(* CoDeSys 2.3.9.59 project: 4.2_Engine_Safety_System20170112.pro *)
(* Libraries: WagoLibTerminalDiag.lib 8.11.10 10:37:48, SYSLIBMEM.LIB 8.11.10 10:37:48, SysLibRtc.lib 8.11.10 10:37:48, Util.lib 26.9.14 11:12:46, WagoLib_CAN_Gateway_02.lib*21.5.19 15:49:18, WagoLibMBX_01.lib*23.7.19 16:23:10, WagoLibMBX_System_01.lib*10.7.18 13:47:36, Standard.lib 8.11.10 10:37:48, SYSLIBCALLBACK.LIB 8.11.10 10:37:48, WagoLibSockets.lib 14.5.12 10:49:54, SysLibSockets.lib 5.5.11 07:22:24, NETVARUDP_LIB_V23.LIB*29.6.15 15:12:14, WagoLibModbus_IP_01.lib*11.2.19 15:41:00, Wago_MBCFG_ETHERNET_01.lib*10.7.18 13:47:36, Wago_MBCFG_COMMON_01.lib*10.7.18 13:47:36 *)

(* PLC configuration (modules and I/O channels)
0750-1504 16 DO 24V DC 0.5A [Type_10_16_Channels] node 0, in %IB36 out %QB36 {INTTypePAAssignment = PLC; INTTypeModule = plugged}
  AT %QX18.0 [BOOLOnX_Q] Ch_1 Digital output
  AT %QX18.1 [BOOLOnX_Q] Ch_2 Digital output
  AT %QX18.2 [BOOLOnX_Q] Ch_3 Digital output
  AT %QX18.3 [BOOLOnX_Q] Ch_4 Digital output
  AT %QX18.4 [BOOLOnX_Q] Ch_5 Digital output
  AT %QX18.5 [BOOLOnX_Q] Ch_6 Digital output
  AT %QX18.6 [BOOLOnX_Q] Ch_7 Digital output
  AT %QX18.7 [BOOLOnX_Q] Ch_8 Digital output
  AT %QX18.8 [BOOLOnX_Q] Ch_9 Digital output
  AT %QX18.9 [BOOLOnX_Q] Ch_10 Digital output
  AT %QX18.10 [BOOLOnX_Q] Ch_11 Digital output
  AT %QX18.11 [BOOLOnX_Q] Ch_12 Digital output
  AT %QX18.12 [BOOLOnX_Q] Ch_13 Digital output
  AT %QX18.13 [BOOLOnX_Q] Ch_14 Digital output
  AT %QX18.14 [BOOLOnX_Q] Ch_15 Digital output
  AT %QX18.15 [BOOLOnX_Q] Ch_16 Digital output
0750-1405 16 DI 24V DC 3.0ms [Type_1_16_Channels] node 1, in %IB36 out %QB36 {INTTypePAAssignment = PLC; INTTypeModule = plugged}
  AT %IX18.0 [BOOLOnX_I] Ch_1 Digital input
  AT %IX18.1 [BOOLOnX_I] Ch_2 Digital input
  AT %IX18.2 [BOOLOnX_I] Ch_3 Digital input
  AT %IX18.3 [BOOLOnX_I] Ch_4 Digital input
  AT %IX18.4 [BOOLOnX_I] Ch_5 Digital input
  AT %IX18.5 [BOOLOnX_I] Ch_6 Digital input
  AT %IX18.6 [BOOLOnX_I] Ch_7 Digital input
  AT %IX18.7 [BOOLOnX_I] Ch_8 Digital input
  AT %IX18.8 [BOOLOnX_I] Ch_9 Digital input
  AT %IX18.9 [BOOLOnX_I] Ch_10 Digital input
  AT %IX18.10 [BOOLOnX_I] Ch_11 Digital input
  AT %IX18.11 [BOOLOnX_I] Ch_12 Digital input
  AT %IX18.12 [BOOLOnX_I] Ch_13 Digital input
  AT %IX18.13 [BOOLOnX_I] Ch_14 Digital input
  AT %IX18.14 [BOOLOnX_I] Ch_15 Digital input
  AT %IX18.15 [BOOLOnX_I] Ch_16 Digital input
0750-1405 16 DI 24V DC 3.0ms [Type_1_16_Channels] node 2, in %IB36 out %QB38 {INTTypePAAssignment = PLC; INTTypeModule = plugged}
  AT %IX19.0 [BOOLOnX_I] Ch_1 Digital input
  AT %IX19.1 [BOOLOnX_I] Ch_2 Digital input
  AT %IX19.2 [BOOLOnX_I] Ch_3 Digital input
  AT %IX19.3 [BOOLOnX_I] Ch_4 Digital input
  AT %IX19.4 [BOOLOnX_I] Ch_5 Digital input
  AT %IX19.5 [BOOLOnX_I] Ch_6 Digital input
  AT %IX19.6 [BOOLOnX_I] Ch_7 Digital input
  AT %IX19.7 [BOOLOnX_I] Ch_8 Digital input
  AT %IX19.8 [BOOLOnX_I] Ch_9 Digital input
  AT %IX19.9 [BOOLOnX_I] Ch_10 Digital input
  AT %IX19.10 [BOOLOnX_I] Ch_11 Digital input
  AT %IX19.11 [BOOLOnX_I] Ch_12 Digital input
  AT %IX19.12 [BOOLOnX_I] Ch_13 Digital input
  AT %IX19.13 [BOOLOnX_I] Ch_14 Digital input
  AT %IX19.14 [BOOLOnX_I] Ch_15 Digital input
  AT %IX19.15 [BOOLOnX_I] Ch_16 Digital input
0750-0404/0000-0003 Frequency Counter 0.1 Hz -100 kHz [Type_4_1_Channels] node 3, in %IB28 out %QB28 {INTTypePAAssignment = PLC; INTTypeModule = plugged}
  AT %IX0.0 [BOOLOnX_I] Frequency measuring range
  AT %IX0.1 [BOOLOnX_I] Frequency measuring range
  AT %IX0.2 [BOOLOnX_I] Status out 1
  AT %IX0.3 [BOOLOnX_I] Status out 2
  AT %IX0.4 [BOOLOnX_I] Tvd Acknowledge
  AT %IX0.5 [BOOLOnX_I] Status Gate input
  AT %IW1 [WORDOnW_I] Frequency Low Word
  AT %IW2 [WORDOnW_I] Frequency High Word
  AT %QX0.0 [BOOLOnX_Q] Acknowledgment frequency range
  AT %QX0.1 [BOOLOnX_Q] Acknowledgment frequency range
  AT %QX0.2 [BOOLOnX_Q] Control out 1
  AT %QX0.3 [BOOLOnX_Q] Control out 2
  AT %QX0.4 [BOOLOnX_Q] Tvd Request
  AT %QW1 [WORDOnW_Q] Watchdog Time
0750-0404/0000-0003 Frequency Counter 0.1 Hz -100 kHz [Type_4_1_Channels] node 4, in %IB28 out %QB28 {INTTypePAAssignment = PLC; INTTypeModule = plugged}
  AT %IX3.0 [BOOLOnX_I] Frequency measuring range
  AT %IX3.1 [BOOLOnX_I] Frequency measuring range
  AT %IX3.2 [BOOLOnX_I] Status out 1
  AT %IX3.3 [BOOLOnX_I] Status out 2
  AT %IX3.4 [BOOLOnX_I] Tvd Acknowledge
  AT %IX3.5 [BOOLOnX_I] Status Gate input
  AT %IW4 [WORDOnW_I] Frequency Low Word
  AT %IW5 [WORDOnW_I] Frequency High Word
  AT %QX3.0 [BOOLOnX_Q] Acknowledgment frequency range
  AT %QX3.1 [BOOLOnX_Q] Acknowledgment frequency range
  AT %QX3.2 [BOOLOnX_Q] Control out 1
  AT %QX3.3 [BOOLOnX_Q] Control out 2
  AT %QX3.4 [BOOLOnX_Q] Tvd Request
  AT %QW4 [WORDOnW_Q] Watchdog Time
0750-0652#08 RS-232/RS-485 Interface adjustable (8 Bytes) [Type_40_1_Channels] node 5, in %IB34 out %QB34 {INTTypePAAssignment = PLC; INTTypeModule = plugged}
  AT %IB12 [BYTEOnB_I] First Byte of 8
  AT %QB12 [BYTEOnB_Q] First Byte of 8
0750-0652#08 RS-232/RS-485 Interface adjustable (8 Bytes) [Type_40_1_Channels] node 6, in %IB40 out %QB40 {INTTypePAAssignment = PLC; INTTypeModule = plugged}
  AT %IB20 [BYTEOnB_I] First Byte of 8
  AT %QB20 [BYTEOnB_Q] First Byte of 8
0750-0652#08 RS-232/RS-485 Interface adjustable (8 Bytes) [Type_40_1_Channels] node 7, in %IB48 out %QB48 {INTTypePAAssignment = PLC; INTTypeModule = plugged}
  AT %IB28 [BYTEOnB_I] First Byte of 8
  AT %QB28 [BYTEOnB_Q] First Byte of 8
Fieldbus variables [FB_VARS] node 1, in %IB0 out %QB0
Flag variables [FLAG_VARS] node 2, in %IB0 out %QB0
Modbus-Master [MB_MASTER] node 3, in %IB0 out %QB0
*)

(* Task configuration *)
TASK MAIN (PRIORITY := 1, INTERVAL := T#20ms);
	PLC_PRG();
END_TASK
TASK MODBUS (PRIORITY := 4, INTERVAL := T#20ms);
	MBCFG_RCS();
END_TASK

(* Global variable list: Global_Variables *)
VAR_GLOBAL

	Slowdown_RPM_Setpoint: REAL;


	ENGINE_SPD1: REAL;(*4~20mA, 6400 -- 32000, or   0 -- 32767*)
	ENGINE_SPD_GRP2: REAL; (*NPN*)

	NO_OF_GEARTEETH_PER_REVOLUTION: REAL;

	(*not used*)
	ENGINE_TURN_AHEAD: REAL;                (*---------------------------------------------think   not  used---------------------------------------------------------*)
	ENGINE_TURN_ASTERN: REAL;		(*---------------------------------------------think   not  used---------------------------------------------------------*)


	SPEED_CMCR: REAL;					(*---------------------------------------------think   not  used---------------------------------------------------------*)

	ENG_STANDSTILL_P: BOOL;


	OVERSPEED_PARAM: REAL;
	OVERSPEED_3135: BOOL; (*from  RCS*)

	ENG_GRP1_WIRE_BROKEN: BOOL;
	ENG_SPD2_WIRE_BROKEN: BOOL;

	STANDSTILL_PARAM: REAL;

	ESS_SPEED_BKP:	REAL;

	(*----SPEED_MEASUREMENT_ESS---------*)
	SPEED_FACTOR_B: REAL; (* Setpoint from HMI *)
	SPEED_FACTOR_C: REAL; (* Setpoint from HMI *)

	ANALOG_SPEED_ESS_HW: REAL; (* From hardware analog channel,address depand on the PLC configration *)	(*SPEED 2*)

	POSITION_HIGHWORD: WORD; (* From hardware analog channel,address depand on the PLC configration *)	(*ESS ENGINE SPEED 1A*)
	POSITION_LOWWORD: WORD; (* From hardware analog channel,address depand on the PLC configration *)		(*ESS ENGINE SPEED 1B*)

	ANALOG_DETECT_SPEED_ESS: REAL;(*speed 2		OUTPUT*)
	NPN_DETECT_SPEED_ESS: INT; (*speed 1			OUTPUT*)

	(*OVERSPEED  HW *)
	ESS_OVERSPEED_HW_P: BOOL;
	(*OVERSPEED  SW *)
	ESS_OVERSPEED_SW_P: BOOL;

	(*OUTPUT*)

	SAFETY_SPD_MEAS_FAILED: BOOL;

	(*send  to  RCS  for  bakcup*)
	ENGINE_TURN_AHEAD_BK: BOOL;
	ENGINE_TURN_ASTERN_BK: BOOL;

	OVERSPEED_NOT_LATCHED: BOOL;

	ENGINE_SPEED_ECR_MAN_CTRL: REAL;
	ENGINE_SPEED_LC_MAN_CTRL: REAL;

	(*-----------------------------SPEED_TO_WATCH------------------------------------*)
	SPEED_AO_MAX:REAL:= 32767;
	SPEED_AO_MIN:REAL:= 0;

	(*-----------------------EMERGENCY STOP -------------------------------------*)
	(*input*)
	BR_EMERG_STOP_SW : BOOL; (*PROESS1004*)
	BR_EMERG_STOP_INDICATOR : BOOL;(*PROESS1030*)
	BR_EMERG_STOP_WIRING_BROKEN: BOOL;

	BR_PORT_WING_EMERG_STOP_SW: BOOL; (*PROESS1005*)
	BR_PORT_WING_EMERG_INDICATOR: BOOL;
	BR_PORT_WING_EMERG_WIRING_BROKEN: BOOL;

	BR_STBD_WING_EMERG_STOP_SW: BOOL;(*PROESS1006*)
	BR_STBD_WING_EMERG_INDICATOR: BOOL;
	BR_STBD_WING_EMERG_WIRING_BROKEN: BOOL;

	ECR_AUT_EMERG_STOP_SW  : BOOL;(*PROESS1012*)
	ECR_AUT_EMERG_STOP_INDICATOR : BOOL;(*PROESS1038*)
	ECR_AUT_EMERG_STOP_SWITCH_WIRING_BROKEN: BOOL;

	ECR_MAN_EMERG_STOP_SW : BOOL;
	ECR_MAN_EMERG_STOP_INDICATOR: BOOL;
	ECR_MAN_EMERG_STOP_SWITCH_WIRING_BROKEN: BOOL;

	LOC_MAN_EMERG_STOP_SW : BOOL;
	LOC_MAN_EMERG_STOP_INDICATOR: BOOL;
	LOC_MAN_EMERG_STOP_SWITCH_WIRING_BROKEN: BOOL;

	(*output*)
	EMERG_STOP: BOOL := FALSE;
	H_BR_ECR_AUT_EMERG_STOP: BOOL;
	EMERG_STOP_BX_7321C: BOOL;


	(*---------------------------------------------INIT_SIGNAL----------------------------------------------------*)
	(***SLOWDOWN SWITCH***)
	(*input*)
	BR_CTRL: BOOL;
	ECR_CTRL_P: BOOL;

	BR_CANCEL_SLD_P: BOOL;
	BR_CENTER_CANCEL_SLD_P: BOOL;
	BR_PORT_CANCEL_SLD_P: BOOL;
	BR_STBD_CANCEL_SLD_P: BOOL;
	ECR_CANCEL_SLD_P: BOOL;


	BR_CANCEL_OMD_SLD_P: BOOL;
	BR_CENTER_CANCEL_OMD_SLD_P: BOOL;
	BR_PORT_CANCEL_OMD_SLD_P: BOOL;
	BR_STBD_CANCEL_OMD_SLD_P: BOOL;
	ECR_CANCEL_OMD_SLD_P: BOOL;

	(*--PORT OR STBD IN CONTROL--*)
	PORT_IN_CONTROL_P: BOOL;
	STBD_IN_CONTROL_P: BOOL;

	(*OMD SLD LAMP  AND  NORMAL SLD LAMP*)
	OMD_SLD_LAMP :BOOL := FALSE;
	NORMAL_SLD_LAMP  :BOOL  :=  FALSE;

	OMD_SLD_SIGN  :BOOL := FALSE;
	NORMAL_SLD_SIGN	:BOOL  := FALSE;

	(*output*)
	OMD_SLD_OVERRIDE: BOOL;
	SLD_OVERRIDE: BOOL;
	(*HMI*)
	H_BR_ECR_AUT_CANCEL_SLD: BOOL;
	H_BR_ECR_AUT_CANCEL_OMD_SLD: BOOL;


	(***RESET SIGNAL***)
	(*input *)
	BR_ECR_RESET_SAFETY_SYSTEM_PUSHB: BOOL;
	RESET_SAFETY_SYSTEM_MAN_BX_7331C: BOOL;


	(*output*)
	RESET_SIGNAL: BOOL;

	(***FLASH FREQUENCY  HZ***)
	(*FLASHER_FREQUENCY: INT := 1;*)
	FLASHER_FREQUENCY: REAL := 1;
	FLASHER_BLINK: BLINK;
	FLASHER_BLINK_TIME: TIME := T#0.5S;

	(***SHUTDOWN OVERRIDE***)
	(*input*)
	BR_SHD_OVERRIDE_SWITCH: BOOL;
	BR_CENTER_SHD_OVERRIDE_SWITCH: BOOL;
	BR_PORT_SHD_OVERRIDE_SWITCH: BOOL;
	BR_STBD_SHD_OVERRIDE_SWITCH: BOOL;
	ECR_AUT_SHD_OVERRIDE: BOOL;


	SHD_OVERRIDE_MAN_BX_7331C: BOOL;

	(*output*)
	SHD_OVERRIDE: BOOL := FALSE;
	(*to HMI*)
	H_BR_ECR_AUT_CANCEL_SHD: BOOL;

	SHD_OVERRIDE_OPTIONAL_SIGN: BOOL;
	SHD_OVERRIDE_BX_7321C: BOOL;
	(*val*)

	ECR_SHD_DYNAMIC_INPUT_TIMER: TON;
	(*ECR shutdown override signal  LOW flag*)
	ECR_SHD_CANCEL_LOW_FLAG: BOOL := FALSE;
	(*dynamic input*)
	ECR_SHD_CANCEL_DYNAMIC_INPUT: BOOL := FALSE;

	CANCELLED_SLOWDOWN_ACTIVED :BOOL;

	(*during the slowdown delay time flag*)
	DURING_SLOWDOWN_DELAY_TIME: BOOL := FALSE;

	(****OVERRIDE BUTTON LAMP****)
	(*TEST LAMP  SIGNAL*)
	ECR_LAMP_TEST_SIGNAL: BOOL := FALSE;
	BR_LAMP_TEST_SIGNAL: BOOL := FALSE;
	PORT_LAMP_TEST_PB: BOOL := FALSE;
	STBD_LAMP_TEST_PB: BOOL := FALSE;

	(*4 test PB o*)
	TEST_PB_SIGNAL: BOOL ;

	(*SLD*)
	BR_CENTER_SLD_LMP_P: BOOL;
	BR_PORT_SLD_LMP_P: BOOL;
	BR_STBD_SLD_LMP_P: BOOL;
	ECR_CANCEL_SLD_LMP_P: BOOL;
	(*OMD SLD*)
	BR_CENTER_OMD_SLD_LMP_P: BOOL;
	BR_PORT_OMD_SLD_LMP_P: BOOL;
	BR_STBD_OMD_SLD_LMP_P: BOOL;
	ECR_CANCEL_OMD_SLD_LMP_P: BOOL;
	(*SHD*)
	BR_CENTER_SHD_LMP_P: BOOL;
	BR_PORT_SHD_LMP_P: BOOL;
	BR_STBD_SHD_LMP_P: BOOL;
	ECR_CANCEL_SHD_LMP_P: BOOL;


	TO_RCS_SHUTDOWN_EXPECTED: BOOL;
	TO_RCS_SHUTDOWN_OVERRIDE: BOOL;
	TO_RCS_OVERSPEED: BOOL;

	BRIDGE_ENGINE_SPEED_METER: REAL;
	BRIDGE_FWP_ENGINE_SPEED_METER: REAL;
	ECR_ENGINE_SPEED_METER: REAL;

	(*----------------------- SLD_SHD_PROCESS-------------------------------------*)
	(*Failure signal*)
	CYL_COOL_WATER_PRESS_INLET_LOW_SHD_P: BOOL; (*PROSSPS1101S*)
	MAIN_BRG_OIL_PRESS_VERY_LOW_SHD_P: BOOL;(*PROSSPS2002S*)
	Thrust_Bearing_Temp_fore_side_HIGH_SHD_P:BOOL;(*PROSSTS4521S*)
	OILMIST_CONCEN_IN_CRANKCASE_HIGH_SLD_P :BOOL;(*PROSSAS2401S*)
	PISTON_COOL_CYL_1_NO_OIL_FLOW_SHD_P :BOOL;(*PROSSFS2521S*)
	PISTON_COOL_CYL_2_NO_OIL_FLOW_SHD_P :BOOL;(*PROSSFS2522S*)
	PISTON_COOL_CYL_3_NO_OIL_FLOW_SHD_P :BOOL;(*PROSSFS2523S*)
	PISTON_COOL_CYL_4_NO_OIL_FLOW_SHD_P :BOOL;(*PROSSFS2524S*)
	PISTON_COOL_CYL_5_NO_OIL_FLOW_SHD_P :BOOL;(*PROSSFS2525S*)
	AIR_SPRING_PRESS_LOW_SHD_P :BOOL;(*PROSSPS4341S*)
	(*OVERSPEED_NOT_LATCHED: BOOL;*)
	UNIC_CRITICAL_FAIL_BX7331C :BOOL;
	UNIC_SLOWDOWN_REQUEST_BX7331C :BOOL;
	(*addition*)
	UNIC_LOAD_LIMIT_IN_GASMODE_BX7331C :BOOL;
	SLD_SIGN_FROM_ALARM_SYSTEM :BOOL;
	(*新增13路AMS降速及其他降速信号过程变量*)
	AMS_MAIN_BRG_OIL_PRESS_LOW_SLD_P :BOOL; (*AMS主机滑油进口压力低降速*)
	AMS_TURBOCHG_BRG_OIL_PRESS_LOW_SLD_P :BOOL; (*AMS增压器滑油进口压力低降速*)
	AMS_AIR_SPRING_PRESS_LOW_SLD_P :BOOL; (*AMS排气阀空气弹簧压力低降速*)
	AMS_TURBOCHG_SPEED_HIGH_SLD_P :BOOL; (*AMS增压器转速高降速*)
	AMS_CYL_COOL_WATER_TEMP_HIGH_SLD_P :BOOL; (*AMS缸套冷却水出口温度高降速*)
	AMS_PISTON_COOL_OIL_TEMP_HIGH_SLD_P :BOOL; (*AMS缸活塞冷却油出口温度高降速*)
	AMS_THRUST_BRG_OIL_TEMP_HIGH_SLD_P :BOOL; (*AMS推力轴承滑油出口温度高降速*)
	AMS_TURBOCHG_OIL_TEMP_HIGH_SLD_P :BOOL; (*AMS增压器滑油出口温度高降速*)
	AMS_CYL_EXHAUST_TEMP_HIGH_SLD_P :BOOL; (*AMS缸排气温度降速*)
	AMS_TURBOCHG_INLET_EXHAUST_TEMP_HIGH_SLD_P :BOOL; (*AMS增压器进口排气温度降速*)
	AMS_SCAV_BOX_FIRE_TEMP_HIGH_SLD_P :BOOL; (*AMS缸扫气箱着火温度高降速*)
	LUBRICATOR_OIL_FLOW_FAIL_SLD_P :BOOL; (*注油器断流降速*)
	GOVERNOR_SYS_FAULT_SLD_P :BOOL; (*调速器系统异常降速*)


	(*time filter,delay*)
	Cyl_cool_Water_PS_1101S_SHD_time_filter :TIME; (*PROESS0014*)
	Cyl_cool_Water_PS_1101S_SHD_time_delay :TIME ;(*PROESS0015*)

	Main_brng_pres_PS2002S_SHD_time_filter: TIME ;(*PROESS0016*)
	Main_brng_pres_PS2002S_SHD_time_delay: TIME ;(*PROESS0017*)

	Main_brng_temp_TS4521S_SHD_time_filter: TIME ;(*PROESS0018*)
	Main_brng_temp_TS4521S_SHD_time_delay: TIME ;(*PROESS0019*)

	Oilmist_AS2401S_SHD_time_filter: TIME;(*PROESS0020*)
	Oilmist_AS2401S_SHD_time_delay: TIME;(*PROESS0021*)

	Piston_cool_Oil_flow_FS25XXS_SHD_time_filter: TIME ;(*PROESS0022*)
	Piston_cool_Oil_flow_FS25XXS_SHD_time_delay: TIME ;(*PROESS0023*)

	Piston_cool_Oil_flow_FS2521S_SHD_time_filter: TIME ;
	Piston_cool_Oil_flow_FS2521S_SHD_time_delay: TIME;

	Piston_cool_Oil_flow_FS2522S_SHD_time_filter: TIME;
	Piston_cool_Oil_flow_FS2522S_SHD_time_delay: TIME;

	Piston_cool_Oil_flow_FS2523S_SHD_time_filter: TIME ;
	Piston_cool_Oil_flow_FS2523S_SHD_time_delay: TIME;

	Piston_cool_Oil_flow_FS2524S_SHD_time_filter: TIME ;
	Piston_cool_Oil_flow_FS2524S_SHD_time_delay: TIME;

	Piston_cool_Oil_flow_FS2525S_SHD_time_filter: TIME ;
	Piston_cool_Oil_flow_FS2525S_SHD_time_delay: TIME ;

	TC_brng_oil_pres_PS2611S_SHD_time_filter: TIME;(*PROESS0024*)
	TC_brng_oil_pres_PS2611S_SHD_time_delay: TIME;(*PROESS0025*)

	Air_spring_pres_PS4341S_SHD_time_filter: TIME ;(*PROESS0026*)
	Air_spring_pres_PS4341S_SHD_time_delay: TIME ;(*PROESS0027*)

	UNIC_critical_fail_SHD_time_filter: TIME ;(*PROESS0028*)
	UNIC_critical_fail_SHD_time_delay: TIME ;(*PROESS0029*)

	UNIC_Slowdown_req_SLD_time_filter: TIME ;(*PROESS0030*)
	UNIC_Slowdown_req_SLD_time_delay: TIME ;(*PROESS0031*)

	UNIC_SLD_DELAY_WITH_GENERATOR_ENGAGED: TIME := t#120s;
	AMS_SLD_DELAY_WITH_GENERATOR_ENGAGED: TIME := t#120s;

	(*addition*)
	UNIC_LOAD_LIMIT_IN_GASMODE_time_filter: TIME;
	UNIC_LOAD_LIMIT_IN_GASMODE_time_delay: TIME ;

	Slowdown_from_AMS_SHD_time_filter :TIME ;
	Slowdown_from_AMS_SHD_time_delay :TIME;
	(*注油器断流降速时间参数，默认滤波3秒*)
	Lubricator_oil_flow_SLD_time_filter :TIME := t#3s; (*注油器断流降速时间滤波*)
	Lubricator_oil_flow_SLD_time_delay :TIME := t#0s; (*注油器断流降速延时*)
	(*调速器故障降速时间参数，默认滤波3秒*)
	Governor_sys_fault_SLD_time_filter :TIME := t#3s; (*调速器系统异常降速时间滤波*)
	Governor_sys_fault_SLD_time_delay :TIME := t#0s; (*调速器系统异常降速延时*)


	(*other input*)
	SHAFT_GENERATOR_ENGAGED_P: BOOL := FALSE;
	OILMIST_CONCENTRATION_IN_CRANDCASE_HIGH :BOOL;

	(*LED Output*)
	CYL_COOL_WATER_INLET_PRESS_LOW: BOOL;
	MAIN_BRG_OIL_PRESS_VERY_LOW: BOOL;
	MAIN_BRG_OIL_TEMP_HIGH: BOOL;
	OIL_CONCENTRATION_IN_CRANKCASE_HIGH: BOOL;
	PISTON_COOL_CYL_1_NO_OIL_FLOW :BOOL;
	PISTON_COOL_CYL_2_NO_OIL_FLOW :BOOL;
	PISTON_COOL_CYL_3_NO_OIL_FLOW :BOOL;
	PISTON_COOL_CYL_4_NO_OIL_FLOW :BOOL;
	PISTON_COOL_CYL_5_NO_OIL_FLOW :BOOL;
	TURBOCHG_1_BRG_OIL_PRESS_LOW :BOOL;
	AIR_SPRING_PRESS_VERY_LOW :BOOL;
	UNIC_CRITICAL_FAIL :BOOL;
	UNIC_SLOWDOWN_REQUEST :BOOL;
	(*addition*)
	UNIC_LOAD_LIMIT_IN_GASMODE :BOOL;
	SLD_MULTIPLE_SOURCE :BOOL;
	(*新增13路降速LED状态输出*)
	AMS_MAIN_BRG_OIL_PRESS_LOW :BOOL; (*AMS主机滑油压力低降速指示*)
	AMS_TURBOCHG_BRG_OIL_PRESS_LOW :BOOL; (*AMS增压器轴承油压低降速指示*)
	AMS_AIR_SPRING_PRESS_LOW :BOOL; (*AMS排气阀弹簧空气压力低降速指示*)
	AMS_TURBOCHG_SPEED_HIGH :BOOL; (*AMS增压器转速高降速指示*)
	AMS_CYL_COOL_WATER_TEMP_HIGH :BOOL; (*AMS缸套冷却水出口温度高降速指示*)
	AMS_PISTON_COOL_OIL_TEMP_HIGH :BOOL; (*AMS缸活塞冷却油出口温度高降速指示*)
	AMS_THRUST_BRG_OIL_TEMP_HIGH :BOOL; (*AMS推力轴承滑油出口温度高降速指示*)
	AMS_TURBOCHG_OIL_TEMP_HIGH :BOOL; (*AMS增压器滑油出口温度高降速指示*)
	AMS_CYL_EXHAUST_TEMP_HIGH :BOOL; (*AMS缸排气温度高降速指示*)
	AMS_TURBOCHG_INLET_EXHAUST_TEMP_HIGH :BOOL; (*AMS增压器进口排气温度高降速指示*)
	AMS_SCAV_BOX_FIRE_TEMP_HIGH :BOOL; (*AMS缸扫气箱着火温度高降速指示*)
	LUBRICATOR_OIL_FLOW_FAIL :BOOL; (*注油器断流降速指示*)
	GOVERNOR_SYS_FAULT :BOOL; (*调速器系统异常降速指示*)

	(*overspeed not latched LAMP output*)
	(*to HMI*)
	H_BR_ECR_AUT_OVERSPEED: BOOL;

	OVERSPEED_BX_7321C :BOOL;

	SLOWDOWN_DURING_GENERATOR_OP_EXPECTED :BOOL;

	(***Page 70.110***)
	(*input*)
	SHUTDOWN_ADR_115: BOOL;(*疑问信号,暂不处理*)
	BR_CEN_ALARM_ACKN_PUSHB : BOOL;
	BR_PORT_ALARM_ACKN_PUSHB : BOOL;
	BR_STBD_ALARM_ACKN_PUSHB : BOOL;
	CR_ALARM_ACKN_PUSHB: BOOL;
	ALARM_ACKN_BX_7331C: BOOL;
	(*output*)
	SLOWDOWN: BOOL;
	SLOWDOWN_ADDR_113: BOOL;(*疑问信号,暂不处理*)
	H_SLOWDOWN_BR_ECR_AUT: BOOL;
	SLD_REQUESTED_BX_7321C: BOOL;
	LOAD_LIMIT_IN_GAS_MODE: BOOL;
	H_LOAD_LIMIT_IN_GAS_MODE_BR_ECR_AUT: BOOL;
	LOAD_LIMIT_IN_GAS_MODE_ACTIVE_BX_7321C: BOOL;
	SHUTDOWN: BOOL;
	H_SHUTDOWN_BR_ECRAUT: BOOL;
	SHD_EXPECTED_BX_7321C: BOOL;
	BR_HORN_ECR_AUT_HORN: BOOL;
	HORN_BX_7321C: BOOL;
	AUX_GEN_REQ: BOOL;(*暂不处理*)

	BR_CEN_ALARM_ACKN_LAMP : BOOL;
	BR_PORT_ALARM_ACKN_LAMP : BOOL;
	BR_STBD_ALARM_ACKN_LAMP : BOOL;
	CR_ALARM_ACKN_LAMP: BOOL;

	SHD_EXPTED_TO_UNIC:	BOOL;
	SLD_EXPTED_TO_UNIC:	BOOL;

	(*--------------------------MISCELLANEOUS-------------------------*)
	(*****input*****)
	Fule_SHD_valve_open_time: TIME := t#60s;
	OPERATION_MODE: BOOL;


	(*WITH PASSIVE FAILURE SUPERVISION*)
	CYL_COOL_WATER_PRESS_INLET_LOW_SHD_PASS_FAIL: BOOL;
	MAIN_BRG_OIL_PRESS_VERY_LOW_SHD_PASS_FAIL: BOOL;
	Thrust_Bearing_Temp_fore_side_HIGH_SHD_PASS_FAIL: BOOL;
	OILMIST_CONCEN_IN_CRANKCASE_HIGH_SLD_PASS_FAIL: BOOL;
	PISTON_COOL_CYL_1_NO_OIL_FLOW_SHD_PASS_FAIL: BOOL;
	PISTON_COOL_CYL_2_NO_OIL_FLOW_SHD_PASS_FAIL: BOOL;
	PISTON_COOL_CYL_3_NO_OIL_FLOW_SHD_PASS_FAIL: BOOL;
	PISTON_COOL_CYL_4_NO_OIL_FLOW_SHD_PASS_FAIL: BOOL;
	PISTON_COOL_CYL_5_NO_OIL_FLOW_SHD_PASS_FAIL: BOOL;
	TURBOCHG_1_BRG_OIL_PRESS_LOW_SHD_PASS_FAIL: BOOL;
	AIR_SPRING_PRESS_LOW_SHD_PASS_FAIL: BOOL;
	FUEL_SHD_PILOT_VALVE_ZV7061S_PASS_FAIL: BOOL;
	SLD_SIGN_FROM_ALARM_SYSTEM_PASS_FAIL: BOOL;
	(*新增13路降速信号被动故障监测（断线检测）*)
	AMS_MAIN_BRG_OIL_PRESS_LOW_SLD_PASS_FAIL :BOOL; (*AMS主机滑油压力低降速断线*)
	AMS_TURBOCHG_BRG_OIL_PRESS_LOW_SLD_PASS_FAIL :BOOL; (*AMS增压器油压低降速断线*)
	AMS_AIR_SPRING_PRESS_LOW_SLD_PASS_FAIL :BOOL; (*AMS排气阀弹簧压力低降速断线*)
	AMS_TURBOCHG_SPEED_HIGH_SLD_PASS_FAIL :BOOL; (*AMS增压器转速高降速断线*)
	AMS_CYL_COOL_WATER_TEMP_HIGH_SLD_PASS_FAIL :BOOL; (*AMS缸套冷却水温度高降速断线*)
	AMS_PISTON_COOL_OIL_TEMP_HIGH_SLD_PASS_FAIL :BOOL; (*AMS活塞冷却油温度高降速断线*)
	AMS_THRUST_BRG_OIL_TEMP_HIGH_SLD_PASS_FAIL :BOOL; (*AMS推力轴承油温高降速断线*)
	AMS_TURBOCHG_OIL_TEMP_HIGH_SLD_PASS_FAIL :BOOL; (*AMS增压器油温高降速断线*)
	AMS_CYL_EXHAUST_TEMP_HIGH_SLD_PASS_FAIL :BOOL; (*AMS缸排气温度高降速断线*)
	AMS_TURBOCHG_INLET_EXHAUST_TEMP_HIGH_SLD_PASS_FAIL :BOOL; (*AMS增压器进口排气温高降速断线*)
	AMS_SCAV_BOX_FIRE_TEMP_HIGH_SLD_PASS_FAIL :BOOL; (*AMS扫气箱着火温高降速断线*)
	LUBRICATOR_OIL_FLOW_FAIL_SLD_PASS_FAIL :BOOL; (*注油器断流降速断线*)
	GOVERNOR_SYS_FAULT_SLD_PASS_FAIL :BOOL; (*调速器故障降速断线*)


	(*系统正常运行标志*)
	SYSTEM_READY_NORMAL: BOOL := TRUE;

	(*****output*****)
	SHD_TO_UNIC_BX7321C: BOOL;
	FUEL_SHD_PILOT_VALVE_ZV7061S: BOOL;
	SAFETY_STOP_P: BOOL;
	SAFETY_STOP_OPTIONAL_SIGN: BOOL;
	SAFETY_SYSTEM_OPERATED: BOOL;
	SAFETY_SYSTEM_OFF_P: BOOL;
	SAFETY_SYSTEM_OFF_FAIL: BOOL;


	(*output*)
	ESS_RESET: BOOL;

	SHIP_MODE_ACTIVE: BOOL;



	(*--------------------------ENGINE_TRIPPED-------------------------*)
	ENGINE_TRIPPED_P: BOOL;


	(*--------------------------------HW IN  HMI OUT INTER  Variable-----------------------------*)
	FUEL_SHD_PILOT_VALVE_ZV_7061S_RELAY_ON: BOOL;

	CommunicationLost: BOOL;(*    both CAN lines are in break *)


	(*750-452  AI 输入模块 0~20mA, 20mA对应32760,  AD_Scale 为32760/20*)
	AD_Scale: WORD := 1638;
	(*750-555  AO 输出模块 4~20mA, 20mA对应32767, DA_Scale 为32767/16*)
	DA_Scale: WORD := 2048;

	(*---------------------------------SWD-----------------------------*)
	RESET_SAFETY_SYSTEM_PB:   BOOL; (*proess0036*)


	(********************************************* HW Signal **********************************************)
	(*-------------------AI-------------------*)
	ESS_ENGINE_SPEED_1B_LOW AT  %IW1: WORD; (*PROSSST5112S*)	
	ESS_ENGINE_SPEED_1A_HIGH AT  %IW2: WORD; (*PROSSST5111S*) 

	ESS_ENGINE_SPEED_2_ANA	AT  %IW51: WORD;    (*PROSSST5104C*)  (*48*)

	(*-------------------AO-------------------*)
	MCR_ENGINE_SPEED_SAFETY_METER: REAL; (*PROESS1001*)
	LOC_E25_ENGINE_SPEED_SAFETY_METER: REAL; (*PROESS1002*)

	(*-------------------DI-------------------*)
	BR_CANCEL_OMD_SLD						   AT	%IX18.2: BOOL;(*DI-1-3*)  
	BR_CANCEL_SLD							   AT	%IX18.3: BOOL;(*DI-1-4*)  
	BR_CANCEL_SHD							   AT	%IX18.4: BOOL;(*DI-1-5*)   
	BR_EMERG_STOP_SWITCH					   AT	%IX18.10: BOOL;(*DI-1-11*)
	ECR_CANCEL_OMD_SLD					       AT	%IX18.7: BOOL;(*DI-1-8*)	
	ECR_CANCEL_SLD							   AT	%IX18.8: BOOL;(*DI-1-9*)  
	ECR_CANCEL_SHD							   AT	%IX18.9: BOOL;(*DI-1-10*)	
	ECR_AUT_EMERG_STOP_SWITCH                  AT   %IX18.11: BOOL;(*DI-1-12*) 
	LOC_EMERG_STOP_SWITCH                      AT   %IX18.12: BOOL;(*DI-1-13*)
	MAIN_BRG_OIL_PRESS_VERY_LOW_SHD			   AT	%IX18.13: BOOL;(*DI-1-14*)
	TURBOCHG_1_BRG_OIL_PRESS_LOW_SHD	       AT	%IX18.14: BOOL;(*DI-1-15*)
	AIR_SPRING_PRESS_LOW_SHD                   AT   %IX18.115: BOOL;(*DI-1-16*)

	AMS_MAIN_BRG_OIL_PRESS_LOW_SLD             AT   %IX19.3: BOOL; (*DI-2-4*)(*AMS主机滑油进口压力低降速反馈*)
	AMS_TURBOCHG_BRG_OIL_PRESS_LOW_SLD         AT   %IX19.4: BOOL; (*DI-2-5*)(*AMS增压器滑油进口压力低降速反馈*)
	CYL_COOL_WATER_PRESS_INLET_LOW_SHD  	   AT   %IX19.5: BOOL;  (*DI-2-6*)  (*50.0*)
	AMS_AIR_SPRING_PRESS_LOW_SLD               AT   %IX19.6: BOOL; (*DI-2-7*)(*AMS排气阀空气弹簧压力低降速反馈*)
	AMS_TURBOCHG_SPEED_HIGH_SLD                AT   %IX19.7: BOOL; (*DI-2-8*)(*AMS增压器转速高降速反馈*)
	AMS_CYL_COOL_WATER_TEMP_HIGH_SLD           AT   %IX19.8: BOOL; (*DI-2-9*)(*AMS缸套冷却水出口温度高降速反馈*)
	AMS_PISTON_COOL_OIL_TEMP_HIGH_SLD          AT   %IX19.9: BOOL; (*DI-2-10*)(*AMS缸活塞冷却油出口温度高降速反馈*)
	AMS_THRUST_BRG_OIL_TEMP_HIGH_SLD           AT   %IX19.10: BOOL; (*DI-2-11*)(*AMS推力轴承滑油出口温度高降速反馈*)
	AMS_TURBOCHG_OIL_TEMP_HIGH_SLD             AT   %IX19.11: BOOL; (*DI-2-12*)(*AMS增压器滑油出口温度高降速反馈*)
	AMS_CYL_EXHAUST_TEMP_HIGH_SLD              AT   %IX19.12: BOOL; (*DI-2-13*)(*AMS缸排气温度降速反馈*)
	AMS_TURBOCHG_INLET_EXHAUST_TEMP_HIGH_SLD   AT   %IX19.13: BOOL; (*DI-2-14*)(*AMS增压器进口排气温度降速反馈*)
	AMS_SCAV_BOX_FIRE_TEMP_HIGH_SLD            AT   %IX19.14: BOOL; (*DI-2-15*)(*AMS缸扫气箱着火温度高降速反馈*)
	Thrust_Bearing_Temp_fore_side_HIGH_SHD	   AT	%IX19.0: BOOL;  (*DI-2-1*)
	OILMIST_CONCEN_IN_CRANKCASE_HIGH_SLD	   AT	%IX19.1: BOOL;  (*DI-2-2*)
	LUBRICATOR_OIL_FLOW_FAIL_SLD               AT   %IX19.2: BOOL; (*DI-2-3*)(*注油器断流降速反馈*)
	GOVERNOR_SYS_FAULT_SLD                     AT   %IX19.15: BOOL; (*      *)(*调速器系统异常报警降速反馈*)		
	
	
 
	ESS_OVERSPEED_HW						AT	%IX53.15: BOOL; (*PROESS1003*)
	PISTON_COOL_CYL_1_NO_OIL_FLOW_SHD			AT	%IX53.8: BOOL;(*PROSSFS2521S*)
	PISTON_COOL_CYL_2_NO_OIL_FLOW_SHD: BOOL;(*PROSSFS2522S*)
	PISTON_COOL_CYL_3_NO_OIL_FLOW_SHD: BOOL;(*PROSSFS2523S*)
	PISTON_COOL_CYL_4_NO_OIL_FLOW_SHD: BOOL;(*PROSSFS2524S*)
	PISTON_COOL_CYL_5_NO_OIL_FLOW_SHD: BOOL;(*PROSSFS2525S*)
	TURBOCHG_1_BRG_OIL_PRESS_LOW_SHD_PS2611S AT %IX54.12: BOOL;(*PROSSPS2611S*)
	BR_PORT_WING_EMERG_STOP_SWITCH: BOOL;(*PROESS1005*)
	BR_STBD_WING_EMERG_STOP_SWITCH: BOOL;(*PROESS1006*)
	SHAFT_GENERATOR_ENGAGED	AT	%IX54.6: BOOL;(*PROESS1019*)	(*51.6*)
	BR_PORT_CANCEL_SLD: BOOL;(*PROESS1020*)
	BR_PORT_CANCEL_OMD_SLD: BOOL;(*PROESS1021*)
	BR_PORT_CANCEL_SHD: BOOL;(*PROESS1023*)
	BR_STBD_CANCEL_SLD: BOOL;(*PROESS1025*)
	BR_STBD_CANCEL_OMD_SLD: BOOL;(*PROESS1026*)
	BR_STBD_CANCEL_SHD: BOOL;(*PROESS1028*)
	Common_SLD_Request_from_AMS AT %IX54.15: BOOL;(*AMSXS9301S*)
	(*新增13路AMS降速及其他降速DI输入，硬件地址待PLC配置时分配*)

	(*新增13路断线检测DI输入，硬件地址待分配*)
	AMS_MAIN_BRG_OIL_PRESS_LOW_SLD_WIRE_BRK : BOOL; (*AMS主机滑油压力低降速断线检测*)
	AMS_TURBOCHG_BRG_OIL_PRESS_LOW_SLD_WIRE_BRK : BOOL; (*AMS增压器油压低降速断线检测*)
	AMS_AIR_SPRING_PRESS_LOW_SLD_WIRE_BRK : BOOL; (*AMS排气阀弹簧压力低降速断线检测*)
	AMS_TURBOCHG_SPEED_HIGH_SLD_WIRE_BRK : BOOL; (*AMS增压器转速高降速断线检测*)
	AMS_CYL_COOL_WATER_TEMP_HIGH_SLD_WIRE_BRK : BOOL; (*AMS缸套冷却水温度高降速断线检测*)
	AMS_PISTON_COOL_OIL_TEMP_HIGH_SLD_WIRE_BRK : BOOL; (*AMS活塞冷却油温度高降速断线检测*)
	AMS_THRUST_BRG_OIL_TEMP_HIGH_SLD_WIRE_BRK : BOOL; (*AMS推力轴承油温高降速断线检测*)
	AMS_TURBOCHG_OIL_TEMP_HIGH_SLD_WIRE_BRK : BOOL; (*AMS增压器油温高降速断线检测*)
	AMS_CYL_EXHAUST_TEMP_HIGH_SLD_WIRE_BRK : BOOL; (*AMS缸排气温度高降速断线检测*)
	AMS_TURBOCHG_INLET_EXHAUST_TEMP_HIGH_SLD_WIRE_BRK : BOOL; (*AMS增压器进口排气温高降速断线检测*)
	AMS_SCAV_BOX_FIRE_TEMP_HIGH_SLD_WIRE_BRK : BOOL; (*AMS扫气箱着火温高降速断线检测*)
	LUBRICATOR_OIL_FLOW_FAIL_SLD_WIRE_BRK : BOOL; (*注油器断流降速断线检测*)
	GOVERNOR_SYS_FAULT_SLD_WIRE_BRK : BOOL; (*调速器故障降速断线检测*)
	(***new add  -12.24----------****)
	HW_FUEL_SHD_PILOT_VALVE_ZV_7061S_RELAY_ON				AT	%IX54.9:  BOOL;


	BR_CEN_ALARM_ACKN_PB				AT	%IX53.14: BOOL;		(*PROESS1085*)	(*50.14*)
	BR_PORT_ALARM_ACKN_PB: BOOL;		(*PROESS1087*)
	BR_STBD_ALARM_ACKN_PB: BOOL;		(*PROESS1088*)
	ECR_ALARM_ACKN_PB					AT	%IX54.3: BOOL;				(*PROESS1086*)	(*51.3*)


	(*WIRE BROKEN*)
	CYL_COOL_WATER_PRESS_INLET_LOW_SHD_WIRE_BRK			AT	%IX53.1: BOOL; (*PROESS1067*)  (*50.1*)
	MAIN_BRG_OIL_PRESS_VERY_LOW_SHD_WIRE_BRK				AT	%IX53.3: BOOL; (*PROESS1068*)
	Thrust_Bearing_Temp_fore_side_HIGH_SHD_WIRE_BRK			AT	%IX53.5: BOOL; 	(*PROESS1069*)
	OILMIST_CONCEN_IN_CRANKCASE_HIGH_SLD_WIRE_BRK			AT	%IX53.7: BOOL;	 (*PROESS1066*)
	PISTON_COOL_CYL_1_NO_OIL_FLOW_SHD_WIRE_BRK				AT	%IX53.9: BOOL; (*PROESS1070*)
	PISTON_COOL_CYL_2_NO_OIL_FLOW_SHD_WIRE_BRK: BOOL; (*PROESS1071*)
	PISTON_COOL_CYL_3_NO_OIL_FLOW_SHD_WIRE_BRK: BOOL; (*PROESS1072*)
	PISTON_COOL_CYL_4_NO_OIL_FLOW_SHD_WIRE_BRK: BOOL; (*PROESS1073*)
	PISTON_COOL_CYL_5_NO_OIL_FLOW_SHD_WIRE_BRK: BOOL; (*PROESS1074*)
	TURBOCHG_1_BRG_OIL_PRESS_LOW_SHD_PS2611S_WIRE_BRK: BOOL; (*PROESS1075*)
	AIR_SPRING_PRESS_LOW_SHD_WIRE_BRK: BOOL; (*PROESS1076*)
	BR_EMERG_STOP_SWITCH_WIRE_BRK									AT	%IX53.11: BOOL; (*PROESS1060*)
	BR_PORT_WING_EMERG_STOP_SWITCH_WIRE_BRK: BOOL; (*PROESS1061*)
	BR_STBD_WING_EMERG_STOP_SWITCH_WIRE_BRK: BOOL; (*PROESS1062*)
	ECR_AUT_EMERG_STOP_SWITCH_WIRE_BRK: BOOL; (*PROESS1063*)
	LOC_EMERG_STOP_SWITCH_WIRE_BRK: BOOL; (*PROESS1064*)
	Common_SLD_Request_from_AMS_WIRE_BRK: BOOL; (*PROESS1065*)
	FUEL_SHD_PILOT_VALVE_DRIVE_WIRE_BRK  AT	%IX55.12 : BOOL; (*PROESS1077*)

	(*-------------------DO-------------------*)
	BR_CANCEL_OMD_SLD_LMP						AT	%QX18.2: BOOL;(*DO-1-3*)  	
	BR_CANCEL_SLD_LMP							AT	%QX18.3: BOOL;(*DO-1-4*)    
	BR_CANCEL_SHD_LMP							AT	%QX18.4: BOOL;(*DO-1-5*)  	
	BR_EMERG_STOP_LMP							AT	%QX18.0: BOOL;(*DO-1-1*)    
	ECR_CANCEL_OMD_SLD_LMP						AT	%QX18.7: BOOL;(*DO-1-8*)	
	ECR_CANCEL_SLD_LMP							AT	%QX18.8: BOOL;(*DO-1-9*)  	
	ECR_CANCEL_SHD_LMP							AT	%QX18.9: BOOL;(*DO-1-10*)	
	ECR_AUT_EMERG_STOP_LMP						AT	%QX18.5: BOOL;(*DO-1-6*)  	
	LOC_EMERG_STOP_LMP							AT	%QX18.10: BOOL;(*DO-1-11*)	
	

	FUEL_SHD_PILOT_VALVE_DRIVE      AT	%QX55.0: BOOL;(*PROSSZV7061S*)
	TO_RCS_SHUTDOWN: BOOL;
	TO_RCS_SLOWDOWN_REQUESTED: BOOL;
	TO_RCS_SLOWDOWN_EXPECTED: BOOL;	

	BR_PORT_WING_EMERG_STOP_LMP: BOOL;(*PROESS1031*)
	BR_STBD_WING_EMERG_STOP_LMP: BOOL;(*PROESS1032*)


	SAFETY_STOP										AT	%QX56.3: BOOL;(*PROESS1045*)  (*--------------------------ESS -> RCS*)	(*	53.3	*)
	SAFETY_SYSTEM_OFF								AT	%QX56.4: BOOL;(*PROESS1046*)	(*	53.4	*)
	BR_PORT_CANCEL_SLD_LMP: BOOL;(*PROESS1047*)
	BR_PORT_CANCEL_OMD_SLD_LMP: BOOL;(*PROESS1048*)

	BR_PORT_CANCEL_SHD_LMP: BOOL;(*PROESS1050*)
	BR_STBD_CANCEL_SLD_LMP: BOOL;(*PROESS1052*)
	BR_STBD_CANCEL_OMD_SLD_LMP: BOOL;(*PROESS1053*)
	BR_STBD_CANCEL_SHD_LMP: BOOL;(*PROESS1055*)
	SHAFT_GENERATOR_EXPECTED_SLD:	BOOL;		(*PROESS1057*)
	Safety_System_Responded_ALM: BOOL;(*PROSSXS9011A*)
	Safety_System_Off_Failure_ALM: BOOL;(*PROSSXS9012A*)
	SAFETY_SYS_SPEED_MEAS_FAILED_ALM: BOOL;(*PROSSXS9013A*)
	SLOW_DOWN_TO_RCS_SPEED			AT	%QX56.15 :BOOL; (*PROESS0005*)   (*--------------------------ESS -> RCS*)

	ESS_ENGINE_TURNING_AHEAD_BKP		AT	%QX56.5: BOOL; (*PROESS1078*)
	ESS_ENGINE_TURNING_ASTERN_BKP	AT	%QX56.6: BOOL; (*PROESS1079*)


	BR_CENT_ALARM_ACKN_INDICATOR					AT	%QX55.9: BOOL;			(*PROESS1089*)	(*	52.9	*)
	BR_PORT_ALARM_ACKN_INDICATOR: BOOL;			(*PROESS1091*)
	BR_STBD_ALARM_ACKN_INDICATOR: BOOL;			(*PROESS1092*)
	ECR_ALARM_ACKN_PB_INDICATOR					AT	%QX55.15: BOOL;			(*PROESS1090*)	(*	52.15	*)


(*********************************************ESS & HMI COMMUNICATION SIGNALS LISTt -------11/08/2016***********************************************)

	  SWD_swd_me_ess_61 AT %QW300: UINT;
	SWD_swd_me_ess_shd_0 AT %QW302: UINT;
	  SC_swd_me_ess_61 AT %IW400: UINT;
	  SCS_swd_me_ess_2_61 AT %QW301: UINT;


	(***HMI ----- > ESS***)

	FRM_BR_CONTROL  :BOOL; 	(*PRORCCAN2001     SP_swd_perm_essout_1_62*)
	FRM_ECR_AUT_CONTROL  :BOOL;  (*PRORCCAN2002 	SP_swd_perm_essout_2_62*)
	FRM_ECR_LAMP_TEST_PB : BOOL;  (*PRORCS0139		SP_swd_perm_essout_3_62*)
	FRM_BR_LAMP_TEST_PB  :BOOL;  (*PRORCS0140		SP_swd_perm_essout_4_62*)
	FRM_PORT_LAMP_TEST_PB :BOOL;  (*PRORCS0141	SP_swd_perm_essout_5_62*)
	FRM_STBD_LAMP_TEST_PB    :BOOL;  (*PRORCS0142	SP_swd_perm_essout_6_62*)
	FRM_OVERSPEED_BKP  :BOOL;      (*PRORCS0001		SP_swd_perm_essout_7_62*)
	FRM_PORT_IN_CONTROL :BOOL;  (*PRORCS9001		SP_swd_perm_essout_8_62*)
	FRM_STBD_IN_CONTROL  :BOOL;  (*PRORCS9002		SP_swd_perm_essout_9_62*)


	(****************ESS--->HMI*********************)
	ESS_ENGINE_SPEED_BKP		AT	%QW256	:REAL; (*PROESS0004*)
	H_ESS_ENGINE_SPEED_1		AT	%QW258	:REAL; (*PROESS0071*)
	H_ESS_ENGINE_SPEED_2		AT	%QW260	:REAL; (*PROESS0074*)



	TRM_ESS_ENGINE_STANDSTILL_BKP  AT   %QX270.0   :BOOL := TRUE; (*PROESS0003         SP_swd_perm_ess1_1_62*)
	H_SHUTDOWN_OVERRIDE_ALARM  AT   %QX270.1   :BOOL := TRUE;  (*PROESS0037    SP_swd_perm_ess1_2_62*)
	H_SLOWDOWN_OVERRIDE_ALARM  AT   %QX270.2   :BOOL := TRUE; (*PROESS0038     SP_swd_perm_ess1_3_62*)
	H_OMD_SLOWDOWN_OVERRIDE_ALARM  AT   %QX270.3   :BOOL := TRUE; (*PROESS0039	SP_swd_perm_ess1_4_62*)
	H_EMERGENCY_STOP_ALARM  AT   %QX270.4   :BOOL; (*PROESS0040	SP_swd_perm_ess1_5_62*)
	H_SLOWDOWN_ALARM  AT   %QX270.5   :BOOL; (*PROESS0041		SP_swd_perm_ess1_6_62*)
	H_SHUTDOWN_ALARM  AT   %QX270.6   :BOOL; (*PROESS0042		SP_swd_perm_ess1_7_62*)
	H_ESS_COMM_TO_UNIC_LOST_FAILURE  AT   %QX270.7  :BOOL; (*PROESS0043	SP_swd_perm_ess1_8_62*)
	H_BRG_CENTER_EMCY_STOP   AT   %QX270.8   :BOOL; (*PROESS0044	SP_swd_perm_ess1_9_62*)
	H_BRG_PORT_EMCY_STOP  AT   %QX270.9   :BOOL; (*PROESS0045	SP_swd_perm_ess1_10_62*)
	H_BRG_STBD_EMCY_STOP  AT   %QX270.10  :BOOL; (*PROESS0046	SP_swd_perm_ess1_11_62*)
	H_MCR_AUTO_EMCY_STOP  AT   %QX270.11   :BOOL; (*PROESS0047	SP_swd_perm_ess1_12_62*)
	H_LOCAL_MAN_EMCY_STOP  AT   %QX270.12   :BOOL; (*PROESS0048		SP_swd_perm_ess1_13_62*)
	H_UNIC_SLD_REQUEST  AT   %QX270.13   :BOOL; (*PROESS0049		SP_swd_perm_ess1_14_62*)
	H_COMMON_SLD_FROM_AMS  AT   %QX270.14   :BOOL; (*PROESS0050	SP_swd_perm_ess1_15_62*)



	H_OILMIST_CONCENTRATION_IN_CRANKCASE_HIGH_SLD  AT   %QX271.0   :BOOL; (*PROESS0051		SP_swd_perm_ess2_1_62*)
	H_CYL_COOL_WATER_PRESS_INLET_LOW_SHD  AT   %QX271.1   :BOOL; (*PROESS0052		SP_swd_perm_ess2_2_62*)
	H_MAIN_BRG_OIL_PRESS_INLET_VERY_LOW_SHD  AT   %QX271.2   :BOOL; (*PROESS0053	SP_swd_perm_ess2_3_62*)
	H_MAIN_BRG_OIL_TEMP_FORE_SIDE_HIGH_SHD  AT   %QX271.3   :BOOL; (*PROESS0054		SP_swd_perm_ess2_4_62*)
	H_PISTON_COOL_OIL_FLOW_MONITORING_CYL_1_SHD  AT   %QX271.4   :BOOL; (*PROESS0055		SP_swd_perm_ess2_5_62*)
	H_PISTON_COOL_OIL_FLOW_MONITORING_CYL_2_SHD  AT   %QX271.5   :BOOL; (*PROESS0056		SP_swd_perm_ess2_6_62*)
	H_PISTON_COOL_OIL_FLOW_MONITORING_CYL_3_SHD  AT   %QX271.6   :BOOL; (*PROESS0057		SP_swd_perm_ess2_7_62*)
	H_PISTON_COOL_OIL_FLOW_MONITORING_CYL_4_SHD  AT   %QX271.7   :BOOL; (*PROESS0058		SP_swd_perm_ess2_8_62*)
	H_PISTON_COOL_OIL_FLOW_MONITORING_CYL_5_SHD  AT   %QX271.8   :BOOL; (*PROESS0059		SP_swd_perm_ess2_9_62*)
	H_TURBOCHG_BRG_1_OIL_PRESS_LOW_SHD  AT   %QX271.9  :BOOL;	 (*PROESS0060		SP_swd_perm_ess2_10_62*)
	H_AIR_SPRING_PRESS_VERY_LOW_SHD  AT   %QX271.10   :BOOL;		 (*PROESS0061		SP_swd_perm_ess2_11_62*)
	H_ESS_OVERSPEED_SW  AT   %QX271.11   :BOOL;					 (*PROESS0062		SP_swd_perm_ess2_12_62*)
	H_UNIC_CRITICAL_FAIL_SHD  AT   %QX271.12   :BOOL;						 (*PROESS0064		SP_swd_perm_ess2_13_62*)
	H_Safety_STOP  AT   %QX271.13   :BOOL;										 (*PROESS0065		SP_swd_perm_ess2_14_62*)



	H_ESS_ENGINE_TURNING_AHEAD  AT   %QX272.0   :BOOL;		 (*PROESS0072		SP_swd_perm_ess3_1_62*)
	H_ESS_ENGINE_TURNING_ASTERN  AT   %QX272.1   :BOOL;	 (*PROESS0073		SP_swd_perm_ess3_2_62*)
	H_ESS_OVERSPEED_HW  AT   %QX272.2   :BOOL;	 (*PROESS0075		SP_swd_perm_ess3_3_62*)
	H_ESS_ENGINE_SPEED_SENSOR_1_WIRE_BROKEN_FAILURE  AT   %QX272.3   :BOOL; (*PROESS0076	SP_swd_perm_ess3_4_62*)
	H_ESS_ENGINE_SPEED_SENSOR_GRP_2_WIRE_BROKEN_FAILURE  AT   %QX272.4   :BOOL; (*PROESS0077	SP_swd_perm_ess3_5_62*)
	H_SHAFT_GENERATOR_EXPECTED_SLD  AT   %QX272.5   :BOOL; (*PROESS0079	SP_swd_perm_ess3_6_62*)
	H_SLD_SHD_HORN_ACOUSTIC_ALARM  AT   %QX272.6   :BOOL; (*PROESS0080		SP_swd_perm_ess3_7_62*)
	H_BRG_CENTER_EMCY_STOP_WIRE_BROKEN_FAILURE  AT   %QX272.7   :BOOL;(*PROESS0081		SP_swd_perm_ess3_8_62*)
	H_BRG_PORT_EMCY_STOP_WIRE_BROKEN_FAILURE  AT   %QX272.8   :BOOL;(*PROESS0082		SP_swd_perm_ess3_9_62*)
	H_BRG_STBD_EMCY_STOP_WIRE_BROKEN_FAILURE  AT   %QX272.9   :BOOL;(*PROESS0083		SP_swd_perm_ess3_10_62*)
	H_MCR_AUTO_EMCY_STOP_WIRE_BROKEN_FAILURE  AT   %QX272.10   :BOOL;(*PROESS0084		SP_swd_perm_ess3_11_62*)
	H_LOCAL_MAN_EMCY_STOP_WIRE_BROKEN_FAILURE  AT   %QX272.11   :BOOL;(*PROESS0085		SP_swd_perm_ess3_12_62*)
	H_COMMON_SLD_FROM_AMS_WIRE_BROKEN_FAILURE  AT   %QX272.12   :BOOL;(*PROESS0086		SP_swd_perm_ess3_13_62*)
	H_OILMIST_CONCENTRATION_IN_CRANKCASE_HIGH_WIRE_BROKEN_FAILURE  AT   %QX272.13  :BOOL;(*PROESS0087		SP_swd_perm_ess3_14_62*)



	H_CYL_COOL_WATER_PRESS_INLET_LOW_WIRE_BROKEN_FAILURE  AT   %QX273.0   :BOOL;(*PROESS0088		SP_swd_perm_ess4_1_62*)
	H_MAIN_BRG_OIL_PRESS_INLET_VERY_LOW_WIRE_BROKEN_FAILURE  AT   %QX273.1   :BOOL;(*PROESS0089		SP_swd_perm_ess4_2_62*)
	H_MAIN_BRG_OIL_TEMP_FORE_SIDE_HIGH_WIRE_BROKEN_FAILURE  AT   %QX273.2   :BOOL;(*PROESS0090		SP_swd_perm_ess4_3_62*)
	H_PISTON_COOL_OIL_FLOW_MONITORING_CYL_1_WIRE_BROKEN_FAILURE  AT   %QX273.3   :BOOL;(*PROESS0091		SP_swd_perm_ess4_4_62*)
	H_PISTON_COOL_OIL_FLOW_MONITORING_CYL_2_WIRE_BROKEN_FAILURE  AT   %QX273.4   :BOOL;(*PROESS0092		SP_swd_perm_ess4_5_62*)
	H_PISTON_COOL_OIL_FLOW_MONITORING_CYL_3_WIRE_BROKEN_FAILURE  AT   %QX273.5   :BOOL;(*PROESS0093		SP_swd_perm_ess4_6_62*)
	H_PISTON_COOL_OIL_FLOW_MONITORING_CYL_4_WIRE_BROKEN_FAILURE  AT   %QX273.6   :BOOL;(*PROESS0094		SP_swd_perm_ess4_7_62*)
	H_PISTON_COOL_OIL_FLOW_MONITORING_CYL_5_WIRE_BROKEN_FAILURE  AT   %QX273.7   :BOOL;(*PROESS0095		SP_swd_perm_ess4_8_62*)
	H_TURBOCHG_BRG_1_OIL_PRESS_LOW_WIRE_BROKEN_FAILURE  AT   %QX273.8   :BOOL;	 (*PROESS0096		SP_swd_perm_ess4_9_62*)
	H_AIR_SPRING_PRESS_VERY_LOW_WIRE_BROKEN_FAILURE  AT   %QX273.9   :BOOL; 	(*PROESS0097		SP_swd_perm_ess4_10_62*)
	H_FUEL_SHD_PILOT_VALVE_ZV_7061S_WIRE_BROKEN_FAILURE  AT   %QX273.10   :BOOL; 	(*PROESS0098		SP_swd_perm_ess4_11_62*)
	H_ESS_CAN1_TO_UNIC_LOST_FAILURE  AT   %QX273.11   :BOOL;	 (*PROESS0099		SP_swd_perm_ess4_12_62*)
	H_ESS_CAN2_TO_UNIC_LOST_FAILURE  AT   %QX273.12   :BOOL; 	(*PROESS0100		SP_swd_perm_ess4_13_62*)
	H_SHIP_MODE_ACTIVE  AT   %QX273.13   :BOOL; (*PROESS101		SP_swd_perm_ess4_14_62*)
	TRM_TEST_MODE_ACTIVE	  AT   %QX273.14   :BOOL; (*PROESS102		SP_swd_perm_ess4_15_62*)


	TRM_Safety_SYSTEM_OFF_FAIL  AT   %QX274.0  :BOOL; 	 		(*PROESS0103		SP_swd_perm_ess5_1_62*)
	H_BR_CEN_ALARM_ACKN_PUSHB  AT   %QX274.1   :BOOL;		(*PROESS0118		SP_swd_perm_ess5_2_62*)
	H_CR_ALARM_ACKN_PUSHB    AT   %QX274.2   :BOOL;	(*PROESS0119		SP_swd_perm_ess5_3_62*)
	H_BR_PORT_ALARM_ACKN_PUSHB   AT   %QX274.3   :BOOL;	(*PROESS0120		SP_swd_perm_ess5_4_62*)
	H_BR_STBD_ALARM_ACKN_PUSHB  AT   %QX274.4   :BOOL;			(*PROESS0121		SP_swd_perm_ess5_5_62*)
	H_ENGINE_TRIPPED  AT   %QX274.5   :BOOL;			(*PROESS0122		SP_swd_perm_ess5_6_62*)

	H_FUEL_SHD_PILOT_VALVE_ZV_7061S_RELAY_ON	AT   %QX274.6: BOOL;   (*PROESS9123	SP_swd_perm_ess5_7_62*)
	H_OVERSPEED_NOT_LATCHED  AT	%QX274.7:  BOOL;	(*PROESS9124	SP_swd_perm_ess5_8_62*)
	H_SHUTDOWN_TO_UNIC AT %QX274.8:BOOL;(*PROESS9725 *)
	H_SLOWDOWN_TO_RCS AT %QX274.9:BOOL;(*PROESS9726 *)


	H_SLD_TIME_COUNT AT %QW289:REAL;(*SLOWDOWN  Delays Remain Time Shown At HMI*)
	H_SHD_TIME_COUNT AT %QW291:REAL;(*SHUTDOWN Delays Remain Time Shown At HMI*)




(*********************************************ESS UNIC----CAN ***********************************************)
	(***ESS--->UNIC  2 Bytes	0x2009**)
	(*bit 0~7*)
	TU_SHUTDOWN_TO_UNIC: BOOL; (*CD_PROSS0010*)
	TU_SHUTDOWN_EXPECTED: BOOL; (*CD_PROSS0012*)
	TU_SHUTDOWN_OVERRIDE: BOOL; (*CD_PROSS0009*)
	TU_SLOWDOWN_REQUESTED: BOOL; (*CD_PROSS0008*)
	TU_OVERSPEED: BOOL; (*CD_PROSS0013*)
	TU_EMERGENCY_STOP: BOOL; (*CD_PROSS0019*)
	TU_HORN: BOOL; (*CD_PROSS0024*)
	TU_LOAD_LIMIT_IN_GAS_MODE_ACTIVE: BOOL;

	(***ESS--->UNIC  2 Bytes	0x2012**)
	TU_Slowdown_RPM_Setpoint: REAL; (*CD_PRORC1029*)


	(***UNIC--->ESS   2 Bytes***)
	(*bit 0~5*)
	FU_RESET_ESS_MANUAL: BOOL; (*PROSSCAN1001*)
	FU_SHUTDOWN_OVERRIDE_MANUAL: BOOL; (*PROSSCAN1002*)
	FU_ALARM_ACKNOWLEDGE_MANUAL: BOOL; (*PROSSCAN1003*)
	FU_UNIC_CRITICAL_FAILURE: BOOL;  (*PROSSCAN1004*)
	FU_UNIC_SLOWDOWN_REQUEST: BOOL; (*PROSSCAN1005*)
	FU_UNIC_LOAD_LIMIT_IN_GAS_MODE: BOOL; (*PROSSCAN1006*)




	BreakDownCAN1:BOOL;
	BreakDownCAN2:BOOL;
END_VAR



VAR_GLOBAL RETAIN
	SPT_air_spr_4341s_shd_t_d	AT	%IW256	:REAL;
	SPT_air_spr_4341S_shd_t_f	AT	%IW258	:REAL;
	SPT_cyl_cw_1101s_shd_t_dl	AT	%IW260	:REAL;
	SPT_cyl_cw_1101s_shd_t_fi		AT	%IW262	:REAL;
	SPT_eng_turn_ahd	AT	%IW264	:REAL;
	SPT_eng_turn_ast	AT	%IW266	:REAL;
	SPT_ess_no_gearteeth_rev	AT	%IW268	:REAL;
	SPT_ess_spd_cmcr_rpm	AT	%IW270	:REAL;				(*---------------------------------------------NOT used   RESERVE---------------------------------------------------------*)
	SPT_ess_fac_b_eng_spd	AT	%IW272	:REAL;
	SPT_ess_fac_c_eng_spd	AT	%IW274	:REAL;
	SPT_ess_flash_frequency	AT	%IW276	:REAL;
	SPT_fuel_shd_v_open_t	AT	%IW278	:REAL;
	SPT_m_brng_2002s_shd_t_dl	AT	%IW280	:REAL;
	SPT_m_brng_2002s_shd_t_fi	AT	%IW282	:REAL;
	SPT_m_brng_4521s_shd_t_fi	AT	%IW284	:REAL;
	SPT_m_brng_4521s_shd_t_dl	AT	%IW286	:REAL;
	SPT_no_testbed_oper_mod	AT	%IW288	:REAL; 	(*0: TESTBED,  1: SHIP*)
	SPT_omist_2401s_shd_dl	AT	%IW290	:REAL;
	SPT_omist_2401s_shd_t_fi	AT	%IW292	:REAL;
	SPT_over_spd	AT	%IW294	:REAL;
	SPT_pstn_fs2501s_dl	AT	%IW296	:REAL;
	SPT_pstn_fs2501s_fi		AT	%IW298	:REAL;
	SPT_sld_frm_ams_shd_t_d	AT	%IW300	:REAL;
	SPT_sld_frm_ams_shd_t_f	AT	%IW302	:REAL;
	SPT_tc_b_o_2611a_shd_t_dl	AT	%IW304	:REAL;
	SPT_tc_b_o_2611s_shd_t_fi		AT	%IW306	:REAL;
	SPT_unic_crit_fal_shd_t_d	AT	%IW308	:REAL;
	SPT_unic_crit_fal_shd_t_f	AT	%IW310	:REAL;
	SPT_unic_sld_req_shd_t_f	AT	%IW312	:REAL;
	SPT_unic_sld_req_shd_t_d	AT	%IW314	:REAL;
	SPT_unic_sld_gen_eng_dl	AT	%IW316	:REAL;
	SPT_ams_sld_gen_eng_dl	AT	%IW318	:REAL;
	SPT_pstn_fs2502s_dl	AT	%IW320	:REAL;
	SPT_pstn_fs2502s_fi		AT	%IW322	:REAL;
	SPT_pstn_fs2503s_dl	AT	%IW324	:REAL;
	SPT_pstn_fs2503s_fi		AT	%IW326	:REAL;
	SPT_pstn_fs2504s_dl	AT	%IW328	:REAL;
	SPT_pstn_fs2504s_fi	   	AT	%IW330	:REAL;
	SPT_pstn_fs2505s_dl	AT	%IW332	:REAL;
	SPT_pstn_fs2505s_fi		AT	%IW334	:REAL;

	SPT_Slowdown_RPM	AT %IW342 :REAL;

	SPT_engine_standstill	AT %IW344 :REAL;

(*2017-5-25------------------------------ *)
	CP_CDPROESSOUT	AT	%IW380	:REAL;
END_VAR

(* Global variable list: Networkmanagement implicit Variables UDP *)
VAR_GLOBAL CONSTANT
	USE_NWVARS_UDP : BOOL := FALSE;
	MAX_NetVarItems_UDP	: INT := 0;
	MAX_NetVarPDO_Rx_UDP	: INT := 0;
	MAX_NetVarPDO_Tx_UDP	: INT := 0;
	MAX_NetVarOD_UDP		: INT := 0;
END_VAR
VAR_GLOBAL
	pNetVarItems_UDP		: ARRAY[0..MAX_NetVarItems_UDP] OF NetVarDataItem_UDP;
	pNetVarPDO_Rx_UDP		: ARRAY[0..MAX_NetVarPDO_Rx_UDP] OF NetVarPDO_Rx_UDP;
	pNetVarPDO_Tx_UDP		: ARRAY[0..MAX_NetVarPDO_Tx_UDP] OF NetVarPDO_Tx_UDP;
	pNetVarOD_UDP			: ARRAY[0..MAX_NetVarOD_UDP] OF NetVarSDO_UDP;
	pNetVarPDO_Rx_Diagnosis_UDP : ARRAY[0..MAX_NetVarPDO_Rx_UDP] OF NetVarUDPDiagStruct;
	pNetVarPDO_Tx_Diagnosis_UDP : ARRAY[0..MAX_NetVarPDO_Tx_UDP] OF NetVarUDPDiagStruct;
END_VAR

(* POU PLC_PRG, ST *)
PROGRAM PLC_PRG
VAR
	(***FUNCTION BLOCK***)
	(*InputProgramValueMapping*)
	InputProgramValueMapping_FUNC: InputProgramValueMapping;
	(*SWD*)
	SWD_FUNC: SWD;
	(*SPEED*)
	SPEED_FUNC: SPEED;
	(*emergency func*)
	EMERGENCY_STOP_FUNC: EMERGENCY_STOP;

	(*停机/降速通道处理，封装于 SLD_SHD_Channels FB*)
	SLD_SHD_CHANNELS_FUNC: SLD_SHD_Channels;

	SWITCHES_ETC_FUNC: SWITCHES_ETC;
	MISCELLANEOUS_FUNC: MISCELLANEOUS;
	OutputProgramValueMapping_FUNC: OutputProgramValueMapping;

	(*ENGINE_TRIPPED*)
	ENGINE_TRIPPED_FUNC:	ENGINE_TRIPPED;


	(***temp val***)
	SLD_LAMP :BOOL := FALSE;
	SHD_LAMP :BOOL := FALSE;
	SLD_SIGN :BOOL := FALSE;
	SHD_SIGN :BOOL := FALSE;
	HORN :BOOL := FALSE;

	(*BR_HORN_ECR_AUT ....SR input*)
	SRIN1: BOOL;
	SRIN2: BOOL;

	SRIns: SR;

	(*BOOT  time*)
	BOOT_DELAY_TIMER: TON;
END_VAR
BOOT_DELAY_TIMER(IN := TRUE, PT := t#1ms);

IF	BOOT_DELAY_TIMER.Q = FALSE
THEN
	RETURN;
END_IF


(****程序临时变量 ****)
(*INIT  VAR*)
SLD_LAMP  := FALSE;
OMD_SLD_LAMP := FALSE;
NORMAL_SLD_LAMP := FALSE;
OMD_SLD_SIGN := FALSE;
NORMAL_SLD_SIGN  :=  FALSE;
SHD_LAMP := FALSE;
SLD_SIGN  := FALSE;
SHD_SIGN := FALSE;
HORN := FALSE;
SRIN1 := FALSE;
SRIN2 := FALSE;


InputProgramValueMapping_FUNC;

SWD_FUNC;

SPEED_FUNC;

EMERGENCY_STOP_FUNC;

SWITCHES_ETC_FUNC;

(*-----------------------SLD_SHD_PROCESS-----------------------*)
SLD_SHD_CHANNELS_FUNC;
SHD_SIGN        := SLD_SHD_CHANNELS_FUNC.SHD_SIGN_OUT;
SLD_SIGN        := SLD_SHD_CHANNELS_FUNC.SLD_SIGN_OUT;
HORN            := SLD_SHD_CHANNELS_FUNC.HORN_OUT;
SHD_LAMP        := SLD_SHD_CHANNELS_FUNC.SHD_LAMP_OUT;
SLD_LAMP        := SLD_SHD_CHANNELS_FUNC.SLD_LAMP_OUT;
OMD_SLD_LAMP    := SLD_SHD_CHANNELS_FUNC.OMD_SLD_LAMP_OUT;
NORMAL_SLD_LAMP := SLD_SHD_CHANNELS_FUNC.NORMAL_SLD_LAMP_OUT;
OMD_SLD_SIGN    := SLD_SHD_CHANNELS_FUNC.OMD_SLD_SIGN_OUT;
NORMAL_SLD_SIGN := SLD_SHD_CHANNELS_FUNC.NORMAL_SLD_SIGN_OUT;


(************ 总信号合成 *******************)
SLOWDOWN := SLD_SIGN;
SHUTDOWN := SHD_SIGN OR EMERG_STOP;
SLOWDOWN_ADDR_113 := SHUTDOWN OR  SLOWDOWN;


(* 本来是发给主机的 *)
SLD_REQUESTED_BX_7321C  :=  SLD_LAMP  OR  SLD_EXPTED_TO_UNIC;
SHD_EXPECTED_BX_7321C  :=  SHD_EXPTED_TO_UNIC;


H_SHUTDOWN_BR_ECRAUT := SHD_EXPECTED_BX_7321C;
H_SLOWDOWN_BR_ECR_AUT := SLD_REQUESTED_BX_7321C;


(*******************蜂鸣报警与报警确认***********************)
SRIN1 := HORN OR EMERG_STOP;
SRIN2 := BR_CEN_ALARM_ACKN_PUSHB
		  OR BR_PORT_ALARM_ACKN_PUSHB
		  OR BR_STBD_ALARM_ACKN_PUSHB
		  OR CR_ALARM_ACKN_PUSHB
		  OR ALARM_ACKN_BX_7331C;

SRIns (SET1 := SRIN1, RESET := SRIN2);
BR_HORN_ECR_AUT_HORN := SRIns.Q1;(*---------------HMI HORN-------------*)
HORN_BX_7321C := BR_HORN_ECR_AUT_HORN;



(************** 试灯功能 ******************)
IF  ECR_LAMP_TEST_SIGNAL = TRUE THEN
	CR_ALARM_ACKN_LAMP := TRUE;
ELSE
	CR_ALARM_ACKN_LAMP := FALSE;
END_IF

IF  BR_LAMP_TEST_SIGNAL = TRUE THEN
	BR_CEN_ALARM_ACKN_LAMP := TRUE;
ELSE
	BR_CEN_ALARM_ACKN_LAMP := FALSE;
END_IF



(*-----------------------------MISCELLANEOUS-----------------------------*)
MISCELLANEOUS_FUNC;


(*-----------------------------ENGINE_TRIPPED-----------------------------*)
ENGINE_TRIPPED_FUNC;


(*-----------------------------OutputProgramValueMapping-----------------------------*)
OutputProgramValueMapping_FUNC;


(*-----------------------------CAN OUT from ESS to UNIC-----------------------------*)
END_PROGRAM

(* POU InputProgramValueMapping, ST *)
FUNCTION_BLOCK InputProgramValueMapping
VAR_INPUT
END_VAR
VAR_OUTPUT
END_VAR
VAR
END_VAR
(*---------------------------------------------------HMI ---> ESS---------------------------------------------------*)
	(***********SET POINT***************)

IF  SPT_ess_no_gearteeth_rev > 0.0
THEN
	Air_spring_pres_PS4341S_SHD_time_delay := REAL_TO_TIME(SPT_air_spr_4341s_shd_t_d) * 1000;(*PROESS0027*)
	Air_spring_pres_PS4341S_SHD_time_filter :=	REAL_TO_TIME(SPT_air_spr_4341S_shd_t_f) * 1000; (*PROESS0026*)

	Cyl_cool_Water_PS_1101S_SHD_time_filter := REAL_TO_TIME(SPT_cyl_cw_1101s_shd_t_fi) * 1000; (*PROESS0014*)
	Cyl_cool_Water_PS_1101S_SHD_time_delay :=  REAL_TO_TIME(SPT_cyl_cw_1101s_shd_t_dl) * 1000; (*PROESS0015*)

	Main_brng_pres_PS2002S_SHD_time_filter := REAL_TO_TIME(SPT_m_brng_2002s_shd_t_fi) * 1000;(*PROESS0016*)
	Main_brng_pres_PS2002S_SHD_time_delay := REAL_TO_TIME(SPT_m_brng_2002s_shd_t_dl) * 1000;(*PROESS0017*)

	Main_brng_temp_TS4521S_SHD_time_filter := REAL_TO_TIME(SPT_m_brng_4521s_shd_t_fi) * 1000; (*PROESS0018*)
	Main_brng_temp_TS4521S_SHD_time_delay := REAL_TO_TIME(SPT_m_brng_4521s_shd_t_dl) * 1000; (*PROESS0019*)

	Oilmist_AS2401S_SHD_time_filter := REAL_TO_TIME(SPT_omist_2401s_shd_t_fi) * 1000; (*PROESS0020*)
	Oilmist_AS2401S_SHD_time_delay := REAL_TO_TIME(SPT_omist_2401s_shd_dl) * 1000; (*PROESS0021*)

	Piston_cool_Oil_flow_FS2521S_SHD_time_filter := REAL_TO_TIME(SPT_pstn_fs2501s_fi) * 1000;
	Piston_cool_Oil_flow_FS2521S_SHD_time_delay := REAL_TO_TIME(SPT_pstn_fs2501s_dl) * 1000;

	Piston_cool_Oil_flow_FS2522S_SHD_time_filter := REAL_TO_TIME(SPT_pstn_fs2502s_fi) * 1000;
	Piston_cool_Oil_flow_FS2522S_SHD_time_delay := REAL_TO_TIME(SPT_pstn_fs2502s_dl) * 1000;

	Piston_cool_Oil_flow_FS2523S_SHD_time_filter := REAL_TO_TIME(SPT_pstn_fs2503s_fi) * 1000;
	Piston_cool_Oil_flow_FS2523S_SHD_time_delay := REAL_TO_TIME(SPT_pstn_fs2503s_dl) * 1000;

	Piston_cool_Oil_flow_FS2524S_SHD_time_filter := REAL_TO_TIME(SPT_pstn_fs2504s_fi) * 1000;
	Piston_cool_Oil_flow_FS2524S_SHD_time_delay := REAL_TO_TIME(SPT_pstn_fs2504s_dl) * 1000;
	
	Piston_cool_Oil_flow_FS2525S_SHD_time_filter := REAL_TO_TIME(SPT_pstn_fs2505s_fi) * 1000;
	Piston_cool_Oil_flow_FS2525S_SHD_time_delay := REAL_TO_TIME(SPT_pstn_fs2505s_dl) * 1000;
	
	Slowdown_from_AMS_SHD_time_filter := REAL_TO_TIME(SPT_sld_frm_ams_shd_t_f) * 1000;
	Slowdown_from_AMS_SHD_time_delay := REAL_TO_TIME(SPT_sld_frm_ams_shd_t_d) * 1000;

	TC_brng_oil_pres_PS2611S_SHD_time_filter := REAL_TO_TIME(SPT_tc_b_o_2611s_shd_t_fi) * 1000;(*PROESS0024*)
	TC_brng_oil_pres_PS2611S_SHD_time_delay := REAL_TO_TIME(SPT_tc_b_o_2611a_shd_t_dl) * 1000;(*PROESS0025*)

	UNIC_critical_fail_SHD_time_filter := REAL_TO_TIME(SPT_unic_crit_fal_shd_t_f) * 1000;(*PROESS0028*)
	UNIC_critical_fail_SHD_time_delay := REAL_TO_TIME(SPT_unic_crit_fal_shd_t_d) * 1000;(*PROESS0029*)

	UNIC_Slowdown_req_SLD_time_filter := REAL_TO_TIME(SPT_unic_sld_req_shd_t_f) * 1000;(*PROESS0030*)
	UNIC_Slowdown_req_SLD_time_delay := REAL_TO_TIME(SPT_unic_sld_req_shd_t_d) * 1000;(*PROESS0031*)

	UNIC_SLD_DELAY_WITH_GENERATOR_ENGAGED := REAL_TO_TIME(SPT_unic_sld_gen_eng_dl) * 1000;
	AMS_SLD_DELAY_WITH_GENERATOR_ENGAGED := REAL_TO_TIME(SPT_ams_sld_gen_eng_dl) * 1000;

	ENGINE_TURN_AHEAD := SPT_eng_turn_ahd;
	ENGINE_TURN_ASTERN := SPT_eng_turn_ast;

	NO_OF_GEARTEETH_PER_REVOLUTION := SPT_ess_no_gearteeth_rev;

	SPEED_CMCR := SPT_ess_spd_cmcr_rpm;

	FLASHER_FREQUENCY := SPT_ess_flash_frequency;

	Fule_SHD_valve_open_time := REAL_TO_TIME(SPT_fuel_shd_v_open_t *1000.0);

	OPERATION_MODE := REAL_TO_BOOL(SPT_no_testbed_oper_mod);

	OVERSPEED_PARAM := SPT_over_spd;

	STANDSTILL_PARAM :=  SPT_engine_standstill;

	SPEED_FACTOR_B := SPT_ess_fac_b_eng_spd;
	SPEED_FACTOR_C := SPT_ess_fac_c_eng_spd;
END_IF

(* ------------------------------------ come from RCS---------------------------CXJ *)

        MODBUS_CONFIGURATION();
      IF   MBCFG_RCS.MBCFG_Error = 0 THEN
	 FRM_BR_CONTROL :=MBCFG_RCS.FRM_BR_CONTROL_cfg;	(*PRORCCAN2001    *)
	FRM_ECR_AUT_CONTROL  :=MBCFG_RCS.FRM_ECR_AUT_CONTROL_cfg   ;  (*PRORCCAN2002 *)
	FRM_ECR_LAMP_TEST_PB :=MBCFG_RCS.FRM_ECR_LAMP_TEST_PB_cfg ;  (*PRORCS0139	*)
	FRM_BR_LAMP_TEST_PB :=MBCFG_RCS.FRM_BR_LAMP_TEST_PB_cfg;  (*PRORCS0140	*)
	FRM_PORT_LAMP_TEST_PB :=MBCFG_RCS.FRM_PORT_LAMP_TEST_PB_cfg;  (*PRORCS0141*)
	FRM_STBD_LAMP_TEST_PB :=MBCFG_RCS.FRM_STBD_LAMP_TEST_PB_cfg;  (*PRORCS0142*)
	FRM_OVERSPEED_BKP :=MBCFG_RCS.FRM_OVERSPEED_BKP_cfg;      (*PRORCS0001*)
	FRM_PORT_IN_CONTROL :=MBCFG_RCS.FRM_PORT_IN_CONTROL_cfg;  (*PRORCS9001*)
	FRM_STBD_IN_CONTROL :=MBCFG_RCS.FRM_STBD_IN_CONTROL_cfg;  (*PRORCS9002	*)
      END_IF


	BR_CTRL := FRM_BR_CONTROL; 						 			   (*PROESS0108			%IX340.0*)
	ECR_CTRL_P := FRM_ECR_AUT_CONTROL;						   (*PROESS0109			%IX340.1*)
	ECR_LAMP_TEST_SIGNAL := FRM_ECR_LAMP_TEST_PB;		   (*PROESS0110			%IX340.2*)
	BR_LAMP_TEST_SIGNAL := FRM_BR_LAMP_TEST_PB;  		          (*PROESS0111			%IX340.3*)
	PORT_LAMP_TEST_PB := FRM_PORT_LAMP_TEST_PB;  			   (*PROESS0112			%IX340.4*)
	STBD_LAMP_TEST_PB := FRM_STBD_LAMP_TEST_PB;  			   (*PROESS0113			%IX340.5*)
	OVERSPEED_3135 := FRM_OVERSPEED_BKP;					   (*PROESS0115			%IX340.6*)
	PORT_IN_CONTROL_P := FRM_PORT_IN_CONTROL;			   (*PROESS0116			%IX340.7*)
	STBD_IN_CONTROL_P := FRM_STBD_IN_CONTROL;			   (*PROESS0117			%IX340.8*)

(*--------------------------------------------HW AI--------------------------------------------*)

	ANALOG_SPEED_ESS_HW :=  WORD_TO_REAL(ESS_ENGINE_SPEED_2_ANA) ; (* From hardware analog channel,address depand on the PLC configration *)
	POSITION_HIGHWORD := ESS_ENGINE_SPEED_1A_HIGH; (* From hardware analog channel,address depand on the PLC configration *)
	POSITION_LOWWORD := ESS_ENGINE_SPEED_1B_LOW; (* From hardware analog channel,address depand on the PLC configration *)


(*--------------------------------------------HW DI--------------------------------------------*)
	(*FAILURE SIGNAL*)
	CYL_COOL_WATER_PRESS_INLET_LOW_SHD_P := CYL_COOL_WATER_PRESS_INLET_LOW_SHD; (*PROSSPS1101S*)
	MAIN_BRG_OIL_PRESS_VERY_LOW_SHD_P := MAIN_BRG_OIL_PRESS_VERY_LOW_SHD;(*PROSSPS2002S*)
	Thrust_Bearing_Temp_fore_side_HIGH_SHD_P := Thrust_Bearing_Temp_fore_side_HIGH_SHD;(*PROSSTS4521S*)
	OILMIST_CONCEN_IN_CRANKCASE_HIGH_SLD_P := OILMIST_CONCEN_IN_CRANKCASE_HIGH_SLD;(*PROSSAS2401S*)
	AIR_SPRING_PRESS_LOW_SHD_P := AIR_SPRING_PRESS_LOW_SHD;(*PROSSPS4341S*)
	SLD_SIGN_FROM_ALARM_SYSTEM := Common_SLD_Request_from_AMS;(*AMSXS9301S*)

	(*EMERG STOP*)
	BR_EMERG_STOP_SW := BR_EMERG_STOP_SWITCH;(*PROESS1004*)
	BR_PORT_WING_EMERG_STOP_SW := BR_PORT_WING_EMERG_STOP_SWITCH;(*PROESS1005*)
	BR_STBD_WING_EMERG_STOP_SW := BR_STBD_WING_EMERG_STOP_SWITCH;(*PROESS1006*)
	ECR_AUT_EMERG_STOP_SW := ECR_AUT_EMERG_STOP_SWITCH;(*PROESS1012*)
	LOC_MAN_EMERG_STOP_SW := LOC_EMERG_STOP_SWITCH;(*PROESS1018*)

	(*SLD OVERRIDE*)
	BR_CENTER_CANCEL_SLD_P := BR_CANCEL_SLD;(*PROESS1007*)
	BR_PORT_CANCEL_SLD_P := BR_PORT_CANCEL_SLD;(*PROESS1020*)
	BR_STBD_CANCEL_SLD_P := BR_STBD_CANCEL_SLD;(*PROESS1025*)

	(*OMD SLD*)
	BR_PORT_CANCEL_OMD_SLD_P := BR_PORT_CANCEL_OMD_SLD;(*PROESS1021*)
	BR_STBD_CANCEL_OMD_SLD_P := BR_STBD_CANCEL_OMD_SLD;(*PROESS1026*)


	ECR_CANCEL_SLD_P := ECR_CANCEL_SLD;(*PROESS1013*)
	ECR_CANCEL_OMD_SLD_P := ECR_CANCEL_OMD_SLD;(*PROESS1014*)
	BR_CENTER_CANCEL_OMD_SLD_P := BR_CANCEL_OMD_SLD;(*PROESS1008*)

	(*SHD OVERRIDE*)
	BR_CENTER_SHD_OVERRIDE_SWITCH := BR_CANCEL_SHD;(*PROESS1011*)
	BR_PORT_SHD_OVERRIDE_SWITCH := BR_PORT_CANCEL_SHD;(*PROESS1023*)
	BR_STBD_SHD_OVERRIDE_SWITCH := BR_STBD_CANCEL_SHD;(*PROESS1028*)

	ECR_AUT_SHD_OVERRIDE := ECR_CANCEL_SHD;(*PROESS1017*)

	SHAFT_GENERATOR_ENGAGED_P := SHAFT_GENERATOR_ENGAGED;(*PROESS1019*)


	BR_CEN_ALARM_ACKN_PUSHB := BR_CEN_ALARM_ACKN_PB;
	BR_PORT_ALARM_ACKN_PUSHB := BR_PORT_ALARM_ACKN_PB;
	BR_STBD_ALARM_ACKN_PUSHB := BR_STBD_ALARM_ACKN_PB;
	CR_ALARM_ACKN_PUSHB := ECR_ALARM_ACKN_PB;

	(***new add  -12.24----------****)
	FUEL_SHD_PILOT_VALVE_ZV_7061S_RELAY_ON := HW_FUEL_SHD_PILOT_VALVE_ZV_7061S_RELAY_ON;

	(*WIRE BROKEN*)
	(*-----------------------------------think  no  used
	ENG_SPD1_WIRE_BROKEN := ESS_ENGINE_SPEED_1_WIRE_BRK; (*PROESS1057*)
	ENG_GRP2_WIRE_BROKEN := ESS_ENGINE_GRP_SPEED_2_WIRE_BRK; (*PROESS1058*)
	*)

	CYL_COOL_WATER_PRESS_INLET_LOW_SHD_PASS_FAIL := CYL_COOL_WATER_PRESS_INLET_LOW_SHD_WIRE_BRK; (*PROESS1060*)
	MAIN_BRG_OIL_PRESS_VERY_LOW_SHD_PASS_FAIL := MAIN_BRG_OIL_PRESS_VERY_LOW_SHD_WIRE_BRK; (*PROESS1061*)
	Thrust_Bearing_Temp_fore_side_HIGH_SHD_PASS_FAIL := Thrust_Bearing_Temp_fore_side_HIGH_SHD_WIRE_BRK; (*PROESS1062*)
	OILMIST_CONCEN_IN_CRANKCASE_HIGH_SLD_PASS_FAIL := OILMIST_CONCEN_IN_CRANKCASE_HIGH_SLD_WIRE_BRK; (*PROESS1063*)
	TURBOCHG_1_BRG_OIL_PRESS_LOW_SHD_PASS_FAIL := TURBOCHG_1_BRG_OIL_PRESS_LOW_SHD_PS2611S_WIRE_BRK; (*PROESS1069*)
	AIR_SPRING_PRESS_LOW_SHD_PASS_FAIL := AIR_SPRING_PRESS_LOW_SHD_WIRE_BRK; (*PROESS1071*)
	FUEL_SHD_PILOT_VALVE_ZV7061S_PASS_FAIL := FUEL_SHD_PILOT_VALVE_DRIVE_WIRE_BRK; (*PROESS1077*)
	SLD_SIGN_FROM_ALARM_SYSTEM_PASS_FAIL := Common_SLD_Request_from_AMS_WIRE_BRK; (*PROESS1076*)
	(*EMERG STOP WIRE BROKEN*)
	BR_EMERG_STOP_WIRING_BROKEN := BR_EMERG_STOP_SWITCH_WIRE_BRK; (*PROESS1078*)
	BR_PORT_WING_EMERG_WIRING_BROKEN := BR_PORT_WING_EMERG_STOP_SWITCH_WIRE_BRK; (*PROESS1072*)
	BR_STBD_WING_EMERG_WIRING_BROKEN := BR_STBD_WING_EMERG_STOP_SWITCH_WIRE_BRK; (*PROESS1073*)
	ECR_AUT_EMERG_STOP_SWITCH_WIRING_BROKEN := ECR_AUT_EMERG_STOP_SWITCH_WIRE_BRK; (*PROESS1074*)
	LOC_MAN_EMERG_STOP_SWITCH_WIRING_BROKEN := LOC_EMERG_STOP_SWITCH_WIRE_BRK; (*PROESS1075*)


	ESS_OVERSPEED_HW_P := ESS_OVERSPEED_HW; (*PROESS1003*)




(*---------------------------------------------------UNIC TO ESS-----CAN---------------------------------------------------*)
	RESET_SAFETY_SYSTEM_MAN_BX_7331C := FU_RESET_ESS_MANUAL; (*PROSSCAN1001*)
	SHD_OVERRIDE_MAN_BX_7331C := FU_SHUTDOWN_OVERRIDE_MANUAL; (*PROSSCAN1002*)
	ALARM_ACKN_BX_7331C := FU_ALARM_ACKNOWLEDGE_MANUAL; (*PROSSCAN1003*)
	UNIC_CRITICAL_FAIL_BX7331C := FU_UNIC_CRITICAL_FAILURE;  (*PROSSCAN1004*)
	UNIC_SLOWDOWN_REQUEST_BX7331C := FU_UNIC_SLOWDOWN_REQUEST; (*PROSSCAN1005*)
	UNIC_LOAD_LIMIT_IN_GASMODE_BX7331C := FU_UNIC_LOAD_LIMIT_IN_GAS_MODE; (*PROSSCAN1006*)


(*--------------------------------------------------RCS  TO  ESS-----MODBUS---------------------------------------------------*)
	(*****FROM RCS TO ESS******)
	Slowdown_RPM_Setpoint := SPT_Slowdown_RPM	;    (*PRORCS0003*)

(*--------------------------------------------新增13路降速DI信号映射--------------------------------------------*)
	(*硬件DI → 过程变量*)
	AMS_MAIN_BRG_OIL_PRESS_LOW_SLD_P := AMS_MAIN_BRG_OIL_PRESS_LOW_SLD; (*AMS主机滑油进口压力低降速*)
	AMS_TURBOCHG_BRG_OIL_PRESS_LOW_SLD_P := AMS_TURBOCHG_BRG_OIL_PRESS_LOW_SLD; (*AMS增压器滑油进口压力低降速*)
	AMS_AIR_SPRING_PRESS_LOW_SLD_P := AMS_AIR_SPRING_PRESS_LOW_SLD; (*AMS排气阀空气弹簧压力低降速*)
	AMS_TURBOCHG_SPEED_HIGH_SLD_P := AMS_TURBOCHG_SPEED_HIGH_SLD; (*AMS增压器转速高降速*)
	AMS_CYL_COOL_WATER_TEMP_HIGH_SLD_P := AMS_CYL_COOL_WATER_TEMP_HIGH_SLD; (*AMS缸套冷却水出口温度高降速*)
	AMS_PISTON_COOL_OIL_TEMP_HIGH_SLD_P := AMS_PISTON_COOL_OIL_TEMP_HIGH_SLD; (*AMS缸活塞冷却油出口温度高降速*)
	AMS_THRUST_BRG_OIL_TEMP_HIGH_SLD_P := AMS_THRUST_BRG_OIL_TEMP_HIGH_SLD; (*AMS推力轴承滑油出口温度高降速*)
	AMS_TURBOCHG_OIL_TEMP_HIGH_SLD_P := AMS_TURBOCHG_OIL_TEMP_HIGH_SLD; (*AMS增压器滑油出口温度高降速*)
	AMS_CYL_EXHAUST_TEMP_HIGH_SLD_P := AMS_CYL_EXHAUST_TEMP_HIGH_SLD; (*AMS缸排气温度降速*)
	AMS_TURBOCHG_INLET_EXHAUST_TEMP_HIGH_SLD_P := AMS_TURBOCHG_INLET_EXHAUST_TEMP_HIGH_SLD; (*AMS增压器进口排气温度降速*)
	AMS_SCAV_BOX_FIRE_TEMP_HIGH_SLD_P := AMS_SCAV_BOX_FIRE_TEMP_HIGH_SLD; (*AMS缸扫气箱着火温度高降速*)
	LUBRICATOR_OIL_FLOW_FAIL_SLD_P := LUBRICATOR_OIL_FLOW_FAIL_SLD; (*注油器断流降速*)
	GOVERNOR_SYS_FAULT_SLD_P := GOVERNOR_SYS_FAULT_SLD; (*调速器系统异常降速*)
	(*断线检测 WIRE_BRK → PASS_FAIL*)
	AMS_MAIN_BRG_OIL_PRESS_LOW_SLD_PASS_FAIL := AMS_MAIN_BRG_OIL_PRESS_LOW_SLD_WIRE_BRK;
	AMS_TURBOCHG_BRG_OIL_PRESS_LOW_SLD_PASS_FAIL := AMS_TURBOCHG_BRG_OIL_PRESS_LOW_SLD_WIRE_BRK;
	AMS_AIR_SPRING_PRESS_LOW_SLD_PASS_FAIL := AMS_AIR_SPRING_PRESS_LOW_SLD_WIRE_BRK;
	AMS_TURBOCHG_SPEED_HIGH_SLD_PASS_FAIL := AMS_TURBOCHG_SPEED_HIGH_SLD_WIRE_BRK;
	AMS_CYL_COOL_WATER_TEMP_HIGH_SLD_PASS_FAIL := AMS_CYL_COOL_WATER_TEMP_HIGH_SLD_WIRE_BRK;
	AMS_PISTON_COOL_OIL_TEMP_HIGH_SLD_PASS_FAIL := AMS_PISTON_COOL_OIL_TEMP_HIGH_SLD_WIRE_BRK;
	AMS_THRUST_BRG_OIL_TEMP_HIGH_SLD_PASS_FAIL := AMS_THRUST_BRG_OIL_TEMP_HIGH_SLD_WIRE_BRK;
	AMS_TURBOCHG_OIL_TEMP_HIGH_SLD_PASS_FAIL := AMS_TURBOCHG_OIL_TEMP_HIGH_SLD_WIRE_BRK;
	AMS_CYL_EXHAUST_TEMP_HIGH_SLD_PASS_FAIL := AMS_CYL_EXHAUST_TEMP_HIGH_SLD_WIRE_BRK;
	AMS_TURBOCHG_INLET_EXHAUST_TEMP_HIGH_SLD_PASS_FAIL := AMS_TURBOCHG_INLET_EXHAUST_TEMP_HIGH_SLD_WIRE_BRK;
	AMS_SCAV_BOX_FIRE_TEMP_HIGH_SLD_PASS_FAIL := AMS_SCAV_BOX_FIRE_TEMP_HIGH_SLD_WIRE_BRK;
	LUBRICATOR_OIL_FLOW_FAIL_SLD_PASS_FAIL := LUBRICATOR_OIL_FLOW_FAIL_SLD_WIRE_BRK;
	GOVERNOR_SYS_FAULT_SLD_PASS_FAIL := GOVERNOR_SYS_FAULT_SLD_WIRE_BRK;
END_FUNCTION_BLOCK

(* POU Configuration/MODBUS_CONFIGURATION, ST *)
PROGRAM MODBUS_CONFIGURATION
VAR                                
END_VAR                            
(*                                 
   <?xml version="1.0" encoding="UTF-16" standalone="yes"?>
<network xml_structure_version="1" xml_feature_version="1">
	<generator_settings minRTUTaskCycleTimeMs="5" minEthaskCycleTimeMs="5" ethSlaveMultiplier="0.1" rtuInterfaceMultiplier="0.1" taskGeneration="false"/>
	<master_interface type="eth" name="" expanded="true">
		<mb_slave comment="Ethernet MR Controller 100MBit 2Port" name="RCS" expanded="true" type="wago" article-no="0750-0882">
			<mb_connection type="eth" transport="UDP" port="502" ip="192.168.1.1" unitid="1" request_delay_ms="0" response_timeout_ms="50"/>
			<service_connection type="eth" ip="192.168.1.1"/>
			<generic_vars comment="" expanded="false"/>
			<pfc_vars comment="" expanded="true">
				<pfc_var name="FRM_BR_CONTROL_cfg" comment="" data_type="BOOL" iec_addr="%QX285.0" expanded="false" mb_access="ro" explicitAccess="false"/>
				<pfc_var name="FRM_ECR_LAMP_TEST_PB_cfg" comment="" data_type="BOOL" iec_addr="%QX288.9" expanded="false" mb_access="ro" explicitAccess="false"/>
				<pfc_var name="FRM_BR_LAMP_TEST_PB_cfg" comment="" data_type="BOOL" iec_addr="%QX288.10" expanded="false" mb_access="ro" explicitAccess="false"/>
				<pfc_var name="FRM_PORT_LAMP_TEST_PB_cfg" comment="" data_type="BOOL" iec_addr="%QX288.11" expanded="false" mb_access="ro" explicitAccess="false"/>
				<pfc_var name="FRM_STBD_LAMP_TEST_PB_cfg" comment="" data_type="BOOL" iec_addr="%QX288.12" expanded="false" mb_access="ro" explicitAccess="false"/>
				<pfc_var name="FRM_OVERSPEED_BKP_cfg" comment="" data_type="BOOL" iec_addr="%QX286.0" expanded="false" mb_access="ro" explicitAccess="false"/>
				<pfc_var name="FRM_ECR_AUT_CONTROL_cfg" comment="" data_type="BOOL" iec_addr="%QX285.1" expanded="false" mb_access="ro" explicitAccess="false"/>
				<pfc_var name="FRM_PORT_IN_CONTROL_cfg" comment="" data_type="BOOL" iec_addr="%QX287.9" expanded="false" mb_access="ro" explicitAccess="false"/>
				<pfc_var name="FRM_STBD_IN_CONTROL_cfg" comment="" data_type="BOOL" iec_addr="%QX287.15" expanded="false" mb_access="ro" explicitAccess="false"/>
				<pfc_var name="SLD_SHD_TIME_COUNT" comment="" data_type="REAL" iec_addr="%QW289" expanded="false" mb_access="ro" explicitAccess="false"/>
			</pfc_vars>
			<k_bus comment="" expanded="false"/>
		</mb_slave>
	</master_interface>
</network>
                              
*)                                 
;                                  
END_PROGRAM

(* POU Generated Code/Ethernet/MBCFG_RCS, ST *)
PROGRAM MBCFG_RCS(* generated by config one prg for each slave *)

VAR_INPUT

END_VAR

VAR_OUTPUT
       FRM_BR_CONTROL_cfg       :    BOOL;       (**) 
       FRM_ECR_LAMP_TEST_PB_cfg       :    BOOL;       (**) 
       FRM_BR_LAMP_TEST_PB_cfg       :    BOOL;       (**) 
       FRM_PORT_LAMP_TEST_PB_cfg       :    BOOL;       (**) 
       FRM_STBD_LAMP_TEST_PB_cfg       :    BOOL;       (**) 
       FRM_OVERSPEED_BKP_cfg       :    BOOL;       (**) 
       FRM_ECR_AUT_CONTROL_cfg       :    BOOL;       (**) 
       FRM_PORT_IN_CONTROL_cfg       :    BOOL;       (**) 
       FRM_STBD_IN_CONTROL_cfg       :    BOOL;       (**) 
       SLD_SHD_TIME_COUNT       :    REAL;       (**) 

    (*--- system variables (read only) ----------------------------------------*)
    MBCFG_IpAddress     :   STRING(11) := '192.168.1.1'; (* address of this slave *)
    MBCFG_Port          :   UINT := 502;               (* IP - Port *)
    MBCFG_UnitID        :   BYTE := 1;             (* MODBUS Unit-Id *)
    MBCFG_TimeOut       :   TIME := t#50ms;           (* Response timeout*)
	MBCFG_RequestDelay  :   TIME  := t#0ms;         (* 0 means no delay *)
    MBCFG_Error         :   MBCFG_eERROR := MBCFG_START_UP;
	MBCFG_LastJob       :   MBCFG_typCOM_JOB;
    (*-------------------------------------------------------------------------*)
END_VAR

{library private}
VAR CONSTANT
    zz_VARIABLECOUNT:   INT := 10; (* number of variables  *)
    zz_JOBCOUNT     :   INT := 2; (* number of jobs *)
END_VAR
VAR

    (*=== VARIABLE LIST ===============================================================================*)
    zz_VariableList :   ARRAY[1..zz_VARIABLECOUNT] OF MBCFG_typVARIABLE :=
    (    DataType        := MBCFG_TYPE_BOOL,
        ByteOrder       := MBCFG_BYTE_ORDER_0,
        BitSize         := 1,
        ptVar           := 0,
        ReadJobIndex    := 1,
        ReadStartBitNo  := 0,
        WriteJobIndex   := 0,
        WriteStartBitNo := 0 ),
    (    DataType        := MBCFG_TYPE_BOOL,
        ByteOrder       := MBCFG_BYTE_ORDER_0,
        BitSize         := 1,
        ptVar           := 0,
        ReadJobIndex    := 1,
        ReadStartBitNo  := 57,
        WriteJobIndex   := 0,
        WriteStartBitNo := 0 ),
    (    DataType        := MBCFG_TYPE_BOOL,
        ByteOrder       := MBCFG_BYTE_ORDER_0,
        BitSize         := 1,
        ptVar           := 0,
        ReadJobIndex    := 1,
        ReadStartBitNo  := 58,
        WriteJobIndex   := 0,
        WriteStartBitNo := 0 ),
    (    DataType        := MBCFG_TYPE_BOOL,
        ByteOrder       := MBCFG_BYTE_ORDER_0,
        BitSize         := 1,
        ptVar           := 0,
        ReadJobIndex    := 1,
        ReadStartBitNo  := 59,
        WriteJobIndex   := 0,
        WriteStartBitNo := 0 ),
    (    DataType        := MBCFG_TYPE_BOOL,
        ByteOrder       := MBCFG_BYTE_ORDER_0,
        BitSize         := 1,
        ptVar           := 0,
        ReadJobIndex    := 1,
        ReadStartBitNo  := 60,
        WriteJobIndex   := 0,
        WriteStartBitNo := 0 ),
    (    DataType        := MBCFG_TYPE_BOOL,
        ByteOrder       := MBCFG_BYTE_ORDER_0,
        BitSize         := 1,
        ptVar           := 0,
        ReadJobIndex    := 1,
        ReadStartBitNo  := 16,
        WriteJobIndex   := 0,
        WriteStartBitNo := 0 ),
    (    DataType        := MBCFG_TYPE_BOOL,
        ByteOrder       := MBCFG_BYTE_ORDER_0,
        BitSize         := 1,
        ptVar           := 0,
        ReadJobIndex    := 1,
        ReadStartBitNo  := 1,
        WriteJobIndex   := 0,
        WriteStartBitNo := 0 ),
    (    DataType        := MBCFG_TYPE_BOOL,
        ByteOrder       := MBCFG_BYTE_ORDER_0,
        BitSize         := 1,
        ptVar           := 0,
        ReadJobIndex    := 1,
        ReadStartBitNo  := 41,
        WriteJobIndex   := 0,
        WriteStartBitNo := 0 ),
    (    DataType        := MBCFG_TYPE_BOOL,
        ByteOrder       := MBCFG_BYTE_ORDER_0,
        BitSize         := 1,
        ptVar           := 0,
        ReadJobIndex    := 1,
        ReadStartBitNo  := 47,
        WriteJobIndex   := 0,
        WriteStartBitNo := 0 ),
    (    DataType        := MBCFG_TYPE_REAL,
        ByteOrder       := MBCFG_BYTE_ORDER_0,
        BitSize         := 32,
        ptVar           := 0,
        ReadJobIndex    := 2,
        ReadStartBitNo  := 0,
        WriteJobIndex   := 0,
        WriteStartBitNo := 0 )

                        ;
    (*=================================================================================================*)

    (*=== JOB LIST ====================================================================================*)
    zz_JobList     :   ARRAY[1..zz_JOBCOUNT] OF MBCFG_typCOM_JOB :=
     (   Functioncode            := 2,
        ReadStartAddress        := 4560,
        ReadQuantity            := 61,
        WriteStartAddress       := 0,
        WriteQuantity           := 0,
        ptReadData              := 0, 
        ptWriteData             := 0 ),
     (   Functioncode            := 4,
        ReadStartAddress        := 289,
        ReadQuantity            := 2,
        WriteStartAddress       := 0,
        WriteQuantity           := 0,
        ptReadData              := 0, 
        ptWriteData             := 0 )

                        ;
    (*=================================================================================================*)

    (*=== DATA FIELDS =================================================================================*)
     zz_DataField_1_Read       :       ARRAY[1..4] OF WORD;
     zz_DataField_2_Read       :       ARRAY[1..2] OF WORD;
	
    (*=================================================================================================*)

    (*=== MODBUS MASTER =====================================*)
    zz_MBCFG_MASTER_ETH :       MBCFG_MASTER_UDP;
    (*=======================================================*)

END_VAR
(*--- for each variable -------------------------*)
   zz_VariableList[1].ptVar := ADR(FRM_BR_CONTROL_cfg);
   zz_VariableList[2].ptVar := ADR(FRM_ECR_LAMP_TEST_PB_cfg);
   zz_VariableList[3].ptVar := ADR(FRM_BR_LAMP_TEST_PB_cfg);
   zz_VariableList[4].ptVar := ADR(FRM_PORT_LAMP_TEST_PB_cfg);
   zz_VariableList[5].ptVar := ADR(FRM_STBD_LAMP_TEST_PB_cfg);
   zz_VariableList[6].ptVar := ADR(FRM_OVERSPEED_BKP_cfg);
   zz_VariableList[7].ptVar := ADR(FRM_ECR_AUT_CONTROL_cfg);
   zz_VariableList[8].ptVar := ADR(FRM_PORT_IN_CONTROL_cfg);
   zz_VariableList[9].ptVar := ADR(FRM_STBD_IN_CONTROL_cfg);
   zz_VariableList[10].ptVar := ADR(SLD_SHD_TIME_COUNT);

(*-----------------------------------------------*)

(*--- for each job -----------------------------------*)
zz_JobList[1].ptReadData   := ADR(zz_DataField_1_Read);
zz_JobList[2].ptReadData   := ADR(zz_DataField_2_Read);

(*----------------------------------------------------*)


(*#### START OF FIXED CODE #####################################*)
zz_MBCFG_MASTER_ETH(	strIpAddress    := MBCFG_IpAddress,                 (* fixed entry     *)
                        uiPort          := MBCFG_Port,                      (* fixed entry     *)
                        bUnitID         := MBCFG_UnitID,                    (* fixed entry     *)
                        tTimeOut        := MBCFG_TimeOut,                   (* fixed entry     *)
                        iVariableCount  := zz_VARIABLECOUNT,
                        ptVariableList  := ADR(zz_VariableList),
                        iJobCount       := zz_JOBCOUNT,
                        ptJobList       := ADR(zz_JobList),
                        tRequestDelay   := MBCFG_RequestDelay,              (* fixed entry     *)
                        eError          => MBCFG_Error,                     (* fixed entry     *)
                        LastJob         => MBCFG_LastJob                    (* fixed entry     *)
                    );
(*##############################################################*)
END_PROGRAM

(* POU SWD, ST *)
FUNCTION_BLOCK SWD
VAR_INPUT
END_VAR
VAR_OUTPUT
END_VAR
VAR
END_VAR
(*----------------SWD_SLD  ----------------------*)

IF  SLD_OVERRIDE  THEN   SWD_swd_me_ess_61 := 7;  (* SLD_OVERRIDE  *)
ELSIF  OMD_SLD_OVERRIDE  THEN   SWD_swd_me_ess_61 := 8;  (* OMD_SLD_OVERRIDE  *)
ELSIF  SLOWDOWN_ADDR_113  THEN   SWD_swd_me_ess_61 := 3;  (* SLOWDOWN  *)
ELSIF  SLD_REQUESTED_BX_7321C THEN   SWD_swd_me_ess_61 := 11;  (* SLD REQUESTED  *)
ELSE   SWD_swd_me_ess_61:=0;(*me slowdown = 0 UKN*)
END_IF;

(*--------------------------------------------------SHD  SWD ---------------------------------------------------------------------------*)

IF   OVERSPEED_NOT_LATCHED  THEN   SWD_swd_me_ess_shd_0 := 5;  (* OVERSPEED  *)
ELSIF  SHD_OVERRIDE  THEN   SWD_swd_me_ess_shd_0 := 2;  (* SHD_OVERRIDE  *)
ELSIF  EMERG_STOP AND NOT SHUTDOWN THEN   SWD_swd_me_ess_shd_0 := 4;  (* EMERG_STOP  *)
ELSIF  SHUTDOWN AND NOT OVERSPEED_NOT_LATCHED   THEN   SWD_swd_me_ess_shd_0:=1;(* SHUTDOWN  *)
ELSIF  SHD_EXPECTED_BX_7321C   THEN   SWD_swd_me_ess_shd_0:=3;(* SHUTDOWN  EXPECTED *)
ELSIF ENGINE_TRIPPED_P   THEN   SWD_swd_me_ess_shd_0:=6;	(*ENGINE  TRIPPED*)
ELSE   SWD_swd_me_ess_shd_0:=0;(*me shutdown = 0 UKN*)
END_IF;

(*------------------------- SCS_swd_me_ess_2_61  Safety System Reset --------------------------------------------*)
IF  NOT ( BR_CTRL  OR  ECR_CTRL_P) THEN       SCS_swd_me_ess_2_61:=1;(*NOT_ALLOWED   1*)
ELSIF    BR_CTRL  OR  ECR_CTRL_P   THEN       SCS_swd_me_ess_2_61:=2;(*ALLOWED  2*)
ELSE                                          SCS_swd_me_ess_2_61:=0;  (*UNKNOWN    0*)
END_IF;

(*SC_swd_me_ess_61   *)
IF     SC_swd_me_ess_61=2     THEN  RESET_SAFETY_SYSTEM_PB:=TRUE ;
ELSIF  SC_swd_me_ess_61=0     THEN  RESET_SAFETY_SYSTEM_PB:=FALSE   ;
ELSE  RESET_SAFETY_SYSTEM_PB:=FALSE;
END_IF;


BR_ECR_RESET_SAFETY_SYSTEM_PUSHB := RESET_SAFETY_SYSTEM_PB;
END_FUNCTION_BLOCK

(* POU SPEED, ST *)
FUNCTION_BLOCK SPEED
VAR_INPUT
END_VAR
VAR_OUTPUT
END_VAR
VAR
	TempSpd: REAL;
	LSKSLD: BOOL;

	SPEED_TO_WATCH_FUNC: SPEED_TO_WATCH;
END_VAR
NO_OF_GEARTEETH_PER_REVOLUTION := 50;
SPEED_MEASUREMENT_ESS ( GEAR_TEETH_PER_REVOLUTION_SETPOINT := REAL_TO_INT(NO_OF_GEARTEETH_PER_REVOLUTION),
									STANDSTILL_SETPOINT := REAL_TO_INT(STANDSTILL_PARAM),
									OVERSPEED_SETPOINT := REAL_TO_INT(OVERSPEED_PARAM));





(***ESS_SPEED_BKP***)
(*转速绝对值0 ~ 150 rpm  待显示表盘量程为 -150 ~ 150 ,4mA 对应-150, 12mA对应0, 24mA对应150 *)

SPEED_TO_WATCH_FUNC (ESS_SPEED_VALUE := SPEED_MEASUREMENT_ESS.SPEED_ESS,
								 EngTurningAST := SPEED_MEASUREMENT_ESS.TURNING_ASTERN_ESS);


ENGINE_SPEED_ECR_MAN_CTRL :=  SPEED_TO_WATCH_FUNC.VALUE;
ENGINE_SPEED_LC_MAN_CTRL :=  SPEED_TO_WATCH_FUNC.VALUE;

ESS_SPEED_BKP :=  SPEED_MEASUREMENT_ESS.SPEED_ESS;
ENGINE_SPD1  :=  NPN_DETECT_SPEED_ESS;
ENGINE_SPD_GRP2  :=  ANALOG_DETECT_SPEED_ESS;


ESS_OVERSPEED_SW_P :=	 SPEED_MEASUREMENT_ESS.OVERSPEED_ESS;
ENGINE_TURN_AHEAD_BK := SPEED_MEASUREMENT_ESS.TURNING_AHEAD_ESS;
ENGINE_TURN_ASTERN_BK := SPEED_MEASUREMENT_ESS.TURNING_ASTERN_ESS;
ENG_STANDSTILL_P := SPEED_MEASUREMENT_ESS.STANDSTILL_ESS;


ENG_GRP1_WIRE_BROKEN  :=  SPEED_MEASUREMENT_ESS.ESS_NPN_SENSER_FAILURE;
ENG_SPD2_WIRE_BROKEN  :=  SPEED_MEASUREMENT_ESS.ESS_ANALOG_SPEED_SENSER_FAILURE;
SAFETY_SPD_MEAS_FAILED :=  ENG_GRP1_WIRE_BROKEN OR  ENG_SPD2_WIRE_BROKEN;


(***OVERSPEED  NOT   LATCHED***)
OVERSPEED_NOT_LATCHED :=  ESS_OVERSPEED_SW_P
									OR  (ESS_OVERSPEED_HW_P  AND  NOT  ENG_SPD2_WIRE_BROKEN)
									OR  OVERSPEED_3135;
END_FUNCTION_BLOCK

(* POU SPEED_TO_WATCH, ST *)
FUNCTION_BLOCK SPEED_TO_WATCH
VAR_INPUT
	ESS_SPEED_VALUE:REAL;
	EngTurningAST: BOOL;
END_VAR
VAR_OUTPUT
	VALUE:INT;
END_VAR
VAR
	K_VALUE: REAL;
	B_VALUE: REAL;
END_VAR
K_VALUE:=(SPEED_AO_MAX  -  SPEED_AO_MIN)/300;
B_VALUE:=SPEED_AO_MAX-150*K_VALUE;


IF  EngTurningAST
THEN  ESS_SPEED_VALUE:=-ESS_SPEED_VALUE;
END_IF;

VALUE:=REAL_TO_INT(ESS_SPEED_VALUE*K_VALUE+B_VALUE);
END_FUNCTION_BLOCK

(* POU SPEED_MEASUREMENT_ESS, ST *)
PROGRAM SPEED_MEASUREMENT_ESS

VAR
	Position_Low: DINT;
	Position_High: DINT;
	Position_Last_Cycle_1000MS: DINT;
	Position_Last_Cycle_50MS: DINT;
	Position: DINT;
	TURNING_AHEAD_ESS_NPN: BOOL;
	TURNING_ASTERN_ESS_NPN: BOOL;
	STANDSTILL_ESS_NPN: BOOL;
	COUNT_DIFF_1000MS: DINT;
	TEETH_COUNTER_FOR_STANDSTILL_LIMIT_PER_MIN: INT;
	TEETH_COUNTER_FOR_STANDSTILL_LIMIT_PER_SEC: INT;
	OUT_OF_STANDSTILL_LIMIT: BOOL;
	BLINK1: BLINK;
	RT1: R_TRIG;
	ACTIVE_1000MS: BOOL;
	temp1: INT;
	temp2: DINT;
	temp3: INT;
	STANDSTILL_ESS_ANALOG: BOOL;
	T1: TON;
	BLINK2: BLINK;
	RT2: R_TRIG;
	ACTIVE_50MS: BOOL;
	TEETH_COUNTER_FOR_OVERSPEED_LIMIT_PER_50MS: INT;
	TEETH_COUNTER_FOR_OVERSPEED_LIMIT_PER_MIN: INT;
	COUNT_DIFF_50MS: DINT;
	ANALOG_DETECT_SPEED_M: REAL;
	COUNT_DECLINE: BOOL;
	COUNT_DIFF_1000MS_ABS: DINT;
	TURNING_ASTERN_ESS_NPN_M: BOOL;
	NPN_DETECT_SPEED_ESS_M: INT;
END_VAR
VAR_INPUT
	GEAR_TEETH_PER_REVOLUTION_SETPOINT: INT; (* Setpoint from HMI *)
	STANDSTILL_SETPOINT: INT; (* Setpoint from HMI *)
	OVERSPEED_SETPOINT: INT; (* Setpoint from HMI *)
END_VAR
VAR_OUTPUT
	ESS_NPN_SENSER_FAILURE: BOOL; (* Health of the RCS NPN speed dectors *)
	ESS_ANALOG_SPEED_SENSER_FAILURE: BOOL; (* Health of the RCS analog speed dector *)
	STANDSTILL_ESS: BOOL;
	TURNING_ASTERN_ESS: BOOL;
	TURNING_AHEAD_ESS: BOOL;
	SPEED_ESS: REAL;
	OVERSPEED_ESS: BOOL; (* Address depand on the PLC configration *) (*SW*)
	REVOLUTION_COUNTER_PULSE: BOOL; (* Address depand on the PLC configration *)
END_VAR
(* ============================================================ *)
(* SPEED_MEASUREMENT_ESS                                        *)
(* Converted from PLCopen XML LD                               *)
(* ============================================================ *)


(* STANDSTILL SETPOINT RPM CONVERT TO TEETH PER SECOND *)

TEETH_COUNTER_FOR_STANDSTILL_LIMIT_PER_MIN :=
    STANDSTILL_SETPOINT *
    GEAR_TEETH_PER_REVOLUTION_SETPOINT;



TEETH_COUNTER_FOR_STANDSTILL_LIMIT_PER_SEC :=
    TEETH_COUNTER_FOR_STANDSTILL_LIMIT_PER_MIN / 30;


(* GET THE COUNT OF TOOTH (POSITION NUMBER) *)

Position_Low := WORD_TO_DWORD(POSITION_HIGHWORD);
Position_High := SHL(Position_Low, 16);
Position := Position_High + WORD_TO_DWORD(POSITION_LOWWORD);


(* MAKE A RISE PULSE FOR EVERY 1000MS *)

BLINK1(
    ENABLE := TRUE,
    TIMELOW := T#0.9S,
    TIMEHIGH := T#0.1S
);

RT1(
    CLK := BLINK1.OUT
);

ACTIVE_1000MS := RT1.Q;


(* COUNT DIFFERENCE *)

IF ACTIVE_1000MS THEN
    COUNT_DIFF_1000MS := Position - Position_Last_Cycle_1000MS;
END_IF;


(* TURNING AHEAD *)
TURNING_AHEAD_ESS_NPN :=
    COUNT_DIFF_1000MS >
    TEETH_COUNTER_FOR_STANDSTILL_LIMIT_PER_SEC;


(* COUNT DECLINE *)
COUNT_DECLINE := COUNT_DIFF_1000MS < 0;


(* ABS COUNT DIFF *)
IF COUNT_DECLINE THEN
    COUNT_DIFF_1000MS_ABS := ABS(COUNT_DIFF_1000MS);
END_IF;


(* TURNING ASTERN *)
TURNING_ASTERN_ESS_NPN_M :=  COUNT_DIFF_1000MS_ABS > TEETH_COUNTER_FOR_STANDSTILL_LIMIT_PER_SEC;

TURNING_ASTERN_ESS_NPN :=  COUNT_DECLINE AND TURNING_ASTERN_ESS_NPN_M;


(* NPN STANDSTILL *)
STANDSTILL_ESS_NPN :=  NOT TURNING_AHEAD_ESS_NPN AND NOT TURNING_ASTERN_ESS_NPN;


(* SAVE POSITION *)
IF ACTIVE_1000MS THEN
    Position_Last_Cycle_1000MS := Position;
END_IF;


(* NPN DETECT SPEED CALCULATE *)
temp2 := COUNT_DIFF_1000MS * 60;
temp3 := DINT_TO_INT(temp2);

NPN_DETECT_SPEED_ESS_M := temp3 / GEAR_TEETH_PER_REVOLUTION_SETPOINT;

NPN_DETECT_SPEED_ESS := ABS(NPN_DETECT_SPEED_ESS_M);


(* ANALOG SPEED SENSOR FAILURE *)

ESS_ANALOG_SPEED_SENSER_FAILURE :=  ANALOG_SPEED_ESS_HW < 6500;


(* ANALOG SPEED SIGNAL CALCULATE *)

IF NOT ESS_ANALOG_SPEED_SENSER_FAILURE THEN

    ANALOG_DETECT_SPEED_M :=
        ANALOG_SPEED_ESS_HW *
        SPEED_FACTOR_B;

    ANALOG_DETECT_SPEED_ESS :=
        ANALOG_DETECT_SPEED_M +
        SPEED_FACTOR_C;

END_IF;


(* IF SENSOR FAILURE, PUT SPEED TO ZERO *)

IF ESS_ANALOG_SPEED_SENSER_FAILURE THEN

    ANALOG_DETECT_SPEED_ESS := 0;

END_IF;


(* ANALOG STANDSTILL *)

temp1 :=
    STANDSTILL_SETPOINT + 1;

STANDSTILL_ESS_ANALOG :=
    ANALOG_DETECT_SPEED_ESS < temp1;


(* NPN SENSOR FAILURE *)

T1(
    IN :=
        NOT ESS_ANALOG_SPEED_SENSER_FAILURE
        AND STANDSTILL_ESS_NPN
        AND NOT STANDSTILL_ESS_ANALOG,

    PT := T#2S
);

ESS_NPN_SENSER_FAILURE :=
    T1.Q;


(* FINAL STANDSTILL *)

STANDSTILL_ESS :=
    NOT ESS_NPN_SENSER_FAILURE
    AND STANDSTILL_ESS_NPN;


(* FINAL DIRECTION *)

TURNING_ASTERN_ESS :=
    NOT ESS_NPN_SENSER_FAILURE
    AND TURNING_ASTERN_ESS_NPN; 

TURNING_AHEAD_ESS :=
    NOT ESS_NPN_SENSER_FAILURE
    AND TURNING_AHEAD_ESS_NPN;


(* SPEED SOURCE SELECT *)

IF NOT ESS_NPN_SENSER_FAILURE THEN

    SPEED_ESS :=
        NPN_DETECT_SPEED_ESS;

END_IF;


IF NOT ESS_ANALOG_SPEED_SENSER_FAILURE
   AND ESS_NPN_SENSER_FAILURE
THEN

    SPEED_ESS :=
        ANALOG_DETECT_SPEED_ESS;

END_IF;


(* OVERSPEED SETPOINT CONVERT TO TEETH PER 50MS *)

TEETH_COUNTER_FOR_OVERSPEED_LIMIT_PER_MIN :=
    OVERSPEED_SETPOINT *
    GEAR_TEETH_PER_REVOLUTION_SETPOINT;

TEETH_COUNTER_FOR_OVERSPEED_LIMIT_PER_50MS :=
    TEETH_COUNTER_FOR_OVERSPEED_LIMIT_PER_MIN /
    1200;


(* MAKE A RISE PULSE FOR EVERY 50MS *)

BLINK2(
    ENABLE := TRUE,
    TIMELOW := T#40MS,
    TIMEHIGH := T#10MS
);

RT2(
    CLK := BLINK2.OUT
);

ACTIVE_50MS :=
    RT2.Q;


(* DETECT OVERSPEED EVERY 50MS *)

IF ACTIVE_50MS THEN

    COUNT_DIFF_50MS :=
        Position -
        Position_Last_Cycle_50MS;

    COUNT_DIFF_50MS :=
        ABS(COUNT_DIFF_50MS);

    OVERSPEED_ESS :=
        COUNT_DIFF_50MS >
        TEETH_COUNTER_FOR_OVERSPEED_LIMIT_PER_50MS;

END_IF;


(* SAVE POSITION EVERY 50MS *)

IF ACTIVE_50MS THEN

    Position_Last_Cycle_50MS :=
        Position;

END_IF;
END_PROGRAM

(* POU EMERGENCY_STOP, ST *)
(*4.1.6.3*)
FUNCTION_BLOCK EMERGENCY_STOP
VAR
END_VAR
VAR_INPUT
END_VAR
VAR_IN_OUT
END_VAR
EMERG_STOP := BR_EMERG_STOP_SW  OR ECR_AUT_EMERG_STOP_SW  OR LOC_MAN_EMERG_STOP_SW;

H_BR_ECR_AUT_EMERG_STOP := EMERG_STOP;
EMERG_STOP_BX_7321C := EMERG_STOP;

(*BUTTON LAMP--------------WIRING BROKEN , LAMP WILL BE LIT OFF*)
BR_EMERG_STOP_INDICATOR := BR_EMERG_STOP_SW;
ECR_AUT_EMERG_STOP_INDICATOR := ECR_AUT_EMERG_STOP_SW;
LOC_MAN_EMERG_STOP_INDICATOR := LOC_MAN_EMERG_STOP_SW;
END_FUNCTION_BLOCK

(* POU SLD_SHD_Channels, ST *)
FUNCTION_BLOCK SLD_SHD_Channels
VAR_OUTPUT
	SHD_SIGN_OUT        : BOOL; (*停车信号*)
	SLD_SIGN_OUT        : BOOL; (*降速信号*)
	HORN_OUT            : BOOL; (*报警蜂鸣*)
	SHD_LAMP_OUT        : BOOL; (*停车指示灯*)
	SLD_LAMP_OUT        : BOOL; (*降速指示灯*)
	OMD_SLD_LAMP_OUT    : BOOL; (*可取消降速指示灯*)
	NORMAL_SLD_LAMP_OUT : BOOL; (*正常降速指示灯*)
	OMD_SLD_SIGN_OUT    : BOOL; (*可取消降速信号*)
	NORMAL_SLD_SIGN_OUT : BOOL; (*正常降速信号*)
END_VAR
VAR
	(*停车通道 SHD_CH_1~6*)
	SHD_CH_1 : SLD_SHD_PROCESS; (*缸套冷却水进口压力低停车 PS1101S*)
	SHD_CH_1_ACTIVE : BOOL;
	SHD_CH_2 : SLD_SHD_PROCESS; (*主机滑油进口压力极低停车 PS2002S，无滤波延时，不可超越*)
	SHD_CH_2_ACTIVE : BOOL;
	SHD_CH_3 : SLD_SHD_PROCESS; (*推力轴承滑油温度高停车 TS4521S*)
	SHD_CH_3_ACTIVE : BOOL;
	SHD_CH_4 : SLD_SHD_PROCESS; (*增压器轴承滑油进口压力低停车 PS2611S*)
	SHD_CH_4_ACTIVE : BOOL;
	SHD_CH_5 : SLD_SHD_PROCESS; (*排气阀弹簧空气进口压力低停车 PS4341S*)
	SHD_CH_5_ACTIVE : BOOL;
	SHD_CH_6 : SLD_SHD_PROCESS; (*超速停车，不可超越*)
	SHD_CH_6_ACTIVE : BOOL;
	(*降速通道 SLD_CH_1~15*)
	SLD_CH_1  : SLD_SHD_PROCESS; (*曲拐箱油雾浓度高降速，可取消 OMD  AS2401S*)
	SLD_CH_1_ACTIVE  : BOOL;
	SLD_CH_2  : SLD_SHD_PROCESS; (*AMS综合降速信号 AMSXS9301S*)
	SLD_CH_2_ACTIVE  : BOOL;
	SLD_CH_3  : SLD_SHD_PROCESS; (*AMS主机滑油进口压力低降速*)
	SLD_CH_3_ACTIVE  : BOOL;
	SLD_CH_4  : SLD_SHD_PROCESS; (*AMS增压器滑油进口压力低降速*)
	SLD_CH_4_ACTIVE  : BOOL;
	SLD_CH_5  : SLD_SHD_PROCESS; (*AMS排气阀空气弹簧压力低降速*)
	SLD_CH_5_ACTIVE  : BOOL;
	SLD_CH_6  : SLD_SHD_PROCESS; (*AMS增压器转速高降速*)
	SLD_CH_6_ACTIVE  : BOOL;
	SLD_CH_7  : SLD_SHD_PROCESS; (*AMS缸套冷却水出口温度高降速*)
	SLD_CH_7_ACTIVE  : BOOL;
	SLD_CH_8  : SLD_SHD_PROCESS; (*AMS缸活塞冷却油出口温度高降速*)
	SLD_CH_8_ACTIVE  : BOOL;
	SLD_CH_9  : SLD_SHD_PROCESS; (*AMS推力轴承滑油出口温度高降速*)
	SLD_CH_9_ACTIVE  : BOOL;
	SLD_CH_10 : SLD_SHD_PROCESS; (*AMS增压器滑油出口温度高降速*)
	SLD_CH_10_ACTIVE : BOOL;
	SLD_CH_11 : SLD_SHD_PROCESS; (*AMS缸排气温度高降速*)
	SLD_CH_11_ACTIVE : BOOL;
	SLD_CH_12 : SLD_SHD_PROCESS; (*AMS增压器进口排气温度高降速*)
	SLD_CH_12_ACTIVE : BOOL;
	SLD_CH_13 : SLD_SHD_PROCESS; (*AMS缸扫气箱着火温度高降速*)
	SLD_CH_13_ACTIVE : BOOL;
	SLD_CH_14 : SLD_SHD_PROCESS; (*注油器断流降速*)
	SLD_CH_14_ACTIVE : BOOL;
	SLD_CH_15 : SLD_SHD_PROCESS; (*调速器系统异常降速*)
	SLD_CH_15_ACTIVE : BOOL;
	(*HMI时间计数临时数组，各通道剩余延时*)
	SHD_TIME_TEMP : ARRAY[0..5]  OF REAL;
	SLD_TIME_TEMP : ARRAY[0..14] OF REAL;
	i : INT;
	j : INT;
	x : BYTE := 0;
	y : BYTE := 0;
	a : BYTE := 0;
	b : BYTE := 0;
	TEMP_SHD_MIN : REAL := 2000000;
	TEMP_SLD_MIN : REAL := 2000000;
END_VAR
(*每周期初始化输出*)
SHD_SIGN_OUT        := FALSE;
SLD_SIGN_OUT        := FALSE;
HORN_OUT            := FALSE;
SHD_LAMP_OUT        := FALSE;
SLD_LAMP_OUT        := FALSE;
OMD_SLD_LAMP_OUT    := FALSE;
NORMAL_SLD_LAMP_OUT := FALSE;
OMD_SLD_SIGN_OUT    := FALSE;
NORMAL_SLD_SIGN_OUT := FALSE;
FOR i := 0 TO 5 DO
	SHD_TIME_TEMP[i] := 2000000;
END_FOR
FOR j := 0 TO 14 DO
	SLD_TIME_TEMP[j] := 2000000;
END_FOR

(*===========停车通道 SHD===========*)

(*SHD_CH_1: 缸套冷却水进口压力低停车 PS1101S*)
SHD_CH_1(FAILURE := CYL_COOL_WATER_PRESS_INLET_LOW_SHD_P AND (NOT CYL_COOL_WATER_PRESS_INLET_LOW_SHD_PASS_FAIL),
				T_FILTER := Cyl_cool_Water_PS_1101S_SHD_time_filter,
				T_DELAY  := Cyl_cool_Water_PS_1101S_SHD_time_delay,
				OVERRIDE := SHD_OVERRIDE);
CYL_COOL_WATER_INLET_PRESS_LOW := SHD_CH_1.LED;
SHD_LAMP_OUT := SHD_LAMP_OUT OR SHD_CH_1.LAMP;
SHD_SIGN_OUT := SHD_SIGN_OUT OR SHD_CH_1.SIGN;
HORN_OUT     := HORN_OUT OR SHD_CH_1.HORN;
SHD_CH_1_ACTIVE := SHD_CH_1.FILTER_FAILURE_OUT;
IF SHD_CH_1_ACTIVE THEN SHD_TIME_TEMP[0] := SHD_CH_1.TIME_COUNT; END_IF

(*SHD_CH_2: 主机滑油进口压力极低停车 PS2002S，无滤波延时，不可超越*)
SHD_CH_2(FAILURE := MAIN_BRG_OIL_PRESS_VERY_LOW_SHD_P AND (NOT MAIN_BRG_OIL_PRESS_VERY_LOW_SHD_PASS_FAIL),
				T_FILTER := t#0s,
				T_DELAY  := t#0s,
				OVERRIDE := FALSE);
MAIN_BRG_OIL_PRESS_VERY_LOW := SHD_CH_2.LED;
SHD_LAMP_OUT := SHD_LAMP_OUT OR SHD_CH_2.LAMP;
SHD_SIGN_OUT := SHD_SIGN_OUT OR SHD_CH_2.SIGN;
HORN_OUT     := HORN_OUT OR SHD_CH_2.HORN;
SHD_CH_2_ACTIVE := SHD_CH_2.FILTER_FAILURE_OUT;
IF SHD_CH_2_ACTIVE THEN SHD_TIME_TEMP[1] := SHD_CH_2.TIME_COUNT; END_IF

(*SHD_CH_3: 推力轴承滑油温度高停车 TS4521S*)
SHD_CH_3(FAILURE := Thrust_Bearing_Temp_fore_side_HIGH_SHD_P AND (NOT Thrust_Bearing_Temp_fore_side_HIGH_SHD_PASS_FAIL),
				T_FILTER := Main_brng_temp_TS4521S_SHD_time_filter,
				T_DELAY  := Main_brng_temp_TS4521S_SHD_time_delay,
				OVERRIDE := SHD_OVERRIDE);
MAIN_BRG_OIL_TEMP_HIGH := SHD_CH_3.LED;
SHD_LAMP_OUT := SHD_LAMP_OUT OR SHD_CH_3.LAMP;
SHD_SIGN_OUT := SHD_SIGN_OUT OR SHD_CH_3.SIGN;
HORN_OUT     := HORN_OUT OR SHD_CH_3.HORN;
SHD_CH_3_ACTIVE := SHD_CH_3.FILTER_FAILURE_OUT;
IF SHD_CH_3_ACTIVE THEN SHD_TIME_TEMP[2] := SHD_CH_3.TIME_COUNT; END_IF

(*SHD_CH_4: 增压器轴承滑油进口压力低停车 PS2611S*)
SHD_CH_4(FAILURE := TURBOCHG_1_BRG_OIL_PRESS_LOW_SHD AND (NOT TURBOCHG_1_BRG_OIL_PRESS_LOW_SHD_PASS_FAIL),
				T_FILTER := TC_brng_oil_pres_PS2611S_SHD_time_filter,
				T_DELAY  := TC_brng_oil_pres_PS2611S_SHD_time_delay,
				OVERRIDE := SHD_OVERRIDE);
TURBOCHG_1_BRG_OIL_PRESS_LOW := SHD_CH_4.LED;
SHD_LAMP_OUT := SHD_LAMP_OUT OR SHD_CH_4.LAMP;
SHD_SIGN_OUT := SHD_SIGN_OUT OR SHD_CH_4.SIGN;
HORN_OUT     := HORN_OUT OR SHD_CH_4.HORN;
SHD_CH_4_ACTIVE := SHD_CH_4.FILTER_FAILURE_OUT;
IF SHD_CH_4_ACTIVE THEN SHD_TIME_TEMP[3] := SHD_CH_4.TIME_COUNT; END_IF

(*SHD_CH_5: 排气阀弹簧空气进口压力低停车 PS4341S*)
SHD_CH_5(FAILURE := AIR_SPRING_PRESS_LOW_SHD_P AND (NOT AIR_SPRING_PRESS_LOW_SHD_PASS_FAIL),
				T_FILTER := Air_spring_pres_PS4341S_SHD_time_filter,
				T_DELAY  := Air_spring_pres_PS4341S_SHD_time_delay,
				OVERRIDE := SHD_OVERRIDE);
AIR_SPRING_PRESS_VERY_LOW := SHD_CH_5.LED;
SHD_LAMP_OUT := SHD_LAMP_OUT OR SHD_CH_5.LAMP;
SHD_SIGN_OUT := SHD_SIGN_OUT OR SHD_CH_5.SIGN;
HORN_OUT     := HORN_OUT OR SHD_CH_5.HORN;
SHD_CH_5_ACTIVE := SHD_CH_5.FILTER_FAILURE_OUT;
IF SHD_CH_5_ACTIVE THEN SHD_TIME_TEMP[4] := SHD_CH_5.TIME_COUNT; END_IF

(*SHD_CH_6: 超速停车，不可超越*)
SHD_CH_6(FAILURE := OVERSPEED_NOT_LATCHED,
				T_FILTER := t#0s,
				T_DELAY  := t#0s,
				OVERRIDE := FALSE);
H_BR_ECR_AUT_OVERSPEED := SHD_CH_6.LAMP;
OVERSPEED_BX_7321C     := H_BR_ECR_AUT_OVERSPEED;
SHD_SIGN_OUT := SHD_SIGN_OUT OR SHD_CH_6.SIGN;
HORN_OUT     := HORN_OUT OR SHD_CH_6.HORN;
SHD_CH_6_ACTIVE := SHD_CH_6.FILTER_FAILURE_OUT;
IF SHD_CH_6_ACTIVE THEN SHD_TIME_TEMP[5] := SHD_CH_6.TIME_COUNT; END_IF

(*===========降速通道 SLD===========*)

(*SLD_CH_1: 曲拐箱油雾浓度高降速，可取消 OMD  AS2401S*)
SLD_CH_1(FAILURE := OILMIST_CONCEN_IN_CRANKCASE_HIGH_SLD_P AND (NOT OILMIST_CONCEN_IN_CRANKCASE_HIGH_SLD_PASS_FAIL),
				T_FILTER := Oilmist_AS2401S_SHD_time_filter,
				T_DELAY  := Oilmist_AS2401S_SHD_time_delay,
				OVERRIDE := OMD_SLD_OVERRIDE);
OIL_CONCENTRATION_IN_CRANKCASE_HIGH := SLD_CH_1.LED;
SLD_LAMP_OUT     := SLD_LAMP_OUT OR SLD_CH_1.LAMP;
SLD_SIGN_OUT     := SLD_SIGN_OUT OR SLD_CH_1.SIGN;
HORN_OUT         := HORN_OUT OR SLD_CH_1.HORN;
OMD_SLD_LAMP_OUT := OMD_SLD_LAMP_OUT OR SLD_CH_1.LAMP;
OMD_SLD_SIGN_OUT := OMD_SLD_SIGN_OUT OR SLD_CH_1.SIGN;
SLD_CH_1_ACTIVE := SLD_CH_1.FILTER_FAILURE_OUT;
IF SLD_CH_1_ACTIVE THEN SLD_TIME_TEMP[0] := SLD_CH_1.TIME_COUNT; END_IF

(*SLD_CH_2: AMS综合降速信号 AMSXS9301S，轴带发电机接合时使用更长延时*)
IF SHAFT_GENERATOR_ENGAGED_P = FALSE THEN
	SLD_CH_2(FAILURE := SLD_SIGN_FROM_ALARM_SYSTEM AND (NOT SLD_SIGN_FROM_ALARM_SYSTEM_PASS_FAIL),
					T_FILTER := Slowdown_from_AMS_SHD_time_filter,
					T_DELAY  := Slowdown_from_AMS_SHD_time_delay,
					OVERRIDE := SLD_OVERRIDE);
ELSE
	SLD_CH_2(FAILURE := SLD_SIGN_FROM_ALARM_SYSTEM AND (NOT SLD_SIGN_FROM_ALARM_SYSTEM_PASS_FAIL),
					T_FILTER := Slowdown_from_AMS_SHD_time_filter,
					T_DELAY  := AMS_SLD_DELAY_WITH_GENERATOR_ENGAGED,
					OVERRIDE := SLD_OVERRIDE);
END_IF
SLD_MULTIPLE_SOURCE  := SLD_CH_2.LED;
SLD_LAMP_OUT         := SLD_LAMP_OUT OR SLD_CH_2.LAMP;
SLD_SIGN_OUT         := SLD_SIGN_OUT OR SLD_CH_2.SIGN;
HORN_OUT             := HORN_OUT OR SLD_CH_2.HORN;
NORMAL_SLD_LAMP_OUT  := NORMAL_SLD_LAMP_OUT OR SLD_CH_2.LAMP;
NORMAL_SLD_SIGN_OUT  := NORMAL_SLD_SIGN_OUT OR SLD_CH_2.SIGN;
SLD_CH_2_ACTIVE := SLD_CH_2.FILTER_FAILURE_OUT;
IF SLD_CH_2_ACTIVE THEN SLD_TIME_TEMP[1] := SLD_CH_2.TIME_COUNT; END_IF

(*SLD_CH_3: AMS主机滑油进口压力低降速*)
SLD_CH_3(FAILURE := AMS_MAIN_BRG_OIL_PRESS_LOW_SLD_P AND (NOT AMS_MAIN_BRG_OIL_PRESS_LOW_SLD_PASS_FAIL),
				T_FILTER := Slowdown_from_AMS_SHD_time_filter,
				T_DELAY  := Slowdown_from_AMS_SHD_time_delay,
				OVERRIDE := SLD_OVERRIDE);
AMS_MAIN_BRG_OIL_PRESS_LOW := SLD_CH_3.LED;
SLD_LAMP_OUT        := SLD_LAMP_OUT OR SLD_CH_3.LAMP;
SLD_SIGN_OUT        := SLD_SIGN_OUT OR SLD_CH_3.SIGN;
HORN_OUT            := HORN_OUT OR SLD_CH_3.HORN;
NORMAL_SLD_LAMP_OUT := NORMAL_SLD_LAMP_OUT OR SLD_CH_3.LAMP;
NORMAL_SLD_SIGN_OUT := NORMAL_SLD_SIGN_OUT OR SLD_CH_3.SIGN;
SLD_CH_3_ACTIVE := SLD_CH_3.FILTER_FAILURE_OUT;
IF SLD_CH_3_ACTIVE THEN SLD_TIME_TEMP[2] := SLD_CH_3.TIME_COUNT; END_IF

(*SLD_CH_4: AMS增压器滑油进口压力低降速*)
SLD_CH_4(FAILURE := AMS_TURBOCHG_BRG_OIL_PRESS_LOW_SLD_P AND (NOT AMS_TURBOCHG_BRG_OIL_PRESS_LOW_SLD_PASS_FAIL),
				T_FILTER := Slowdown_from_AMS_SHD_time_filter,
				T_DELAY  := Slowdown_from_AMS_SHD_time_delay,
				OVERRIDE := SLD_OVERRIDE);
AMS_TURBOCHG_BRG_OIL_PRESS_LOW := SLD_CH_4.LED;
SLD_LAMP_OUT        := SLD_LAMP_OUT OR SLD_CH_4.LAMP;
SLD_SIGN_OUT        := SLD_SIGN_OUT OR SLD_CH_4.SIGN;
HORN_OUT            := HORN_OUT OR SLD_CH_4.HORN;
NORMAL_SLD_LAMP_OUT := NORMAL_SLD_LAMP_OUT OR SLD_CH_4.LAMP;
NORMAL_SLD_SIGN_OUT := NORMAL_SLD_SIGN_OUT OR SLD_CH_4.SIGN;
SLD_CH_4_ACTIVE := SLD_CH_4.FILTER_FAILURE_OUT;
IF SLD_CH_4_ACTIVE THEN SLD_TIME_TEMP[3] := SLD_CH_4.TIME_COUNT; END_IF

(*SLD_CH_5: AMS排气阀空气弹簧压力低降速*)
SLD_CH_5(FAILURE := AMS_AIR_SPRING_PRESS_LOW_SLD_P AND (NOT AMS_AIR_SPRING_PRESS_LOW_SLD_PASS_FAIL),
				T_FILTER := Slowdown_from_AMS_SHD_time_filter,
				T_DELAY  := Slowdown_from_AMS_SHD_time_delay,
				OVERRIDE := SLD_OVERRIDE);
AMS_AIR_SPRING_PRESS_LOW := SLD_CH_5.LED;
SLD_LAMP_OUT        := SLD_LAMP_OUT OR SLD_CH_5.LAMP;
SLD_SIGN_OUT        := SLD_SIGN_OUT OR SLD_CH_5.SIGN;
HORN_OUT            := HORN_OUT OR SLD_CH_5.HORN;
NORMAL_SLD_LAMP_OUT := NORMAL_SLD_LAMP_OUT OR SLD_CH_5.LAMP;
NORMAL_SLD_SIGN_OUT := NORMAL_SLD_SIGN_OUT OR SLD_CH_5.SIGN;
SLD_CH_5_ACTIVE := SLD_CH_5.FILTER_FAILURE_OUT;
IF SLD_CH_5_ACTIVE THEN SLD_TIME_TEMP[4] := SLD_CH_5.TIME_COUNT; END_IF

(*SLD_CH_6: AMS增压器转速高降速*)
SLD_CH_6(FAILURE := AMS_TURBOCHG_SPEED_HIGH_SLD_P AND (NOT AMS_TURBOCHG_SPEED_HIGH_SLD_PASS_FAIL),
				T_FILTER := Slowdown_from_AMS_SHD_time_filter,
				T_DELAY  := Slowdown_from_AMS_SHD_time_delay,
				OVERRIDE := SLD_OVERRIDE);
AMS_TURBOCHG_SPEED_HIGH := SLD_CH_6.LED;
SLD_LAMP_OUT        := SLD_LAMP_OUT OR SLD_CH_6.LAMP;
SLD_SIGN_OUT        := SLD_SIGN_OUT OR SLD_CH_6.SIGN;
HORN_OUT            := HORN_OUT OR SLD_CH_6.HORN;
NORMAL_SLD_LAMP_OUT := NORMAL_SLD_LAMP_OUT OR SLD_CH_6.LAMP;
NORMAL_SLD_SIGN_OUT := NORMAL_SLD_SIGN_OUT OR SLD_CH_6.SIGN;
SLD_CH_6_ACTIVE := SLD_CH_6.FILTER_FAILURE_OUT;
IF SLD_CH_6_ACTIVE THEN SLD_TIME_TEMP[5] := SLD_CH_6.TIME_COUNT; END_IF

(*SLD_CH_7: AMS缸套冷却水出口温度高降速*)
SLD_CH_7(FAILURE := AMS_CYL_COOL_WATER_TEMP_HIGH_SLD_P AND (NOT AMS_CYL_COOL_WATER_TEMP_HIGH_SLD_PASS_FAIL),
				T_FILTER := Slowdown_from_AMS_SHD_time_filter,
				T_DELAY  := Slowdown_from_AMS_SHD_time_delay,
				OVERRIDE := SLD_OVERRIDE);
AMS_CYL_COOL_WATER_TEMP_HIGH := SLD_CH_7.LED;
SLD_LAMP_OUT        := SLD_LAMP_OUT OR SLD_CH_7.LAMP;
SLD_SIGN_OUT        := SLD_SIGN_OUT OR SLD_CH_7.SIGN;
HORN_OUT            := HORN_OUT OR SLD_CH_7.HORN;
NORMAL_SLD_LAMP_OUT := NORMAL_SLD_LAMP_OUT OR SLD_CH_7.LAMP;
NORMAL_SLD_SIGN_OUT := NORMAL_SLD_SIGN_OUT OR SLD_CH_7.SIGN;
SLD_CH_7_ACTIVE := SLD_CH_7.FILTER_FAILURE_OUT;
IF SLD_CH_7_ACTIVE THEN SLD_TIME_TEMP[6] := SLD_CH_7.TIME_COUNT; END_IF

(*SLD_CH_8: AMS缸活塞冷却油出口温度高降速*)
SLD_CH_8(FAILURE := AMS_PISTON_COOL_OIL_TEMP_HIGH_SLD_P AND (NOT AMS_PISTON_COOL_OIL_TEMP_HIGH_SLD_PASS_FAIL),
				T_FILTER := Slowdown_from_AMS_SHD_time_filter,
				T_DELAY  := Slowdown_from_AMS_SHD_time_delay,
				OVERRIDE := SLD_OVERRIDE);
AMS_PISTON_COOL_OIL_TEMP_HIGH := SLD_CH_8.LED;
SLD_LAMP_OUT        := SLD_LAMP_OUT OR SLD_CH_8.LAMP;
SLD_SIGN_OUT        := SLD_SIGN_OUT OR SLD_CH_8.SIGN;
HORN_OUT            := HORN_OUT OR SLD_CH_8.HORN;
NORMAL_SLD_LAMP_OUT := NORMAL_SLD_LAMP_OUT OR SLD_CH_8.LAMP;
NORMAL_SLD_SIGN_OUT := NORMAL_SLD_SIGN_OUT OR SLD_CH_8.SIGN;
SLD_CH_8_ACTIVE := SLD_CH_8.FILTER_FAILURE_OUT;
IF SLD_CH_8_ACTIVE THEN SLD_TIME_TEMP[7] := SLD_CH_8.TIME_COUNT; END_IF


(*SLD_CH_9: AMS推力轴承滑油出口温度高降速*)
SLD_CH_9(FAILURE := AMS_THRUST_BRG_OIL_TEMP_HIGH_SLD_P AND (NOT AMS_THRUST_BRG_OIL_TEMP_HIGH_SLD_PASS_FAIL),
				T_FILTER := Slowdown_from_AMS_SHD_time_filter,
				T_DELAY  := Slowdown_from_AMS_SHD_time_delay,
				OVERRIDE := SLD_OVERRIDE);
AMS_THRUST_BRG_OIL_TEMP_HIGH := SLD_CH_9.LED;
SLD_LAMP_OUT        := SLD_LAMP_OUT OR SLD_CH_9.LAMP;
SLD_SIGN_OUT        := SLD_SIGN_OUT OR SLD_CH_9.SIGN;
HORN_OUT            := HORN_OUT OR SLD_CH_9.HORN;
NORMAL_SLD_LAMP_OUT := NORMAL_SLD_LAMP_OUT OR SLD_CH_9.LAMP;
NORMAL_SLD_SIGN_OUT := NORMAL_SLD_SIGN_OUT OR SLD_CH_9.SIGN;
SLD_CH_9_ACTIVE := SLD_CH_9.FILTER_FAILURE_OUT;
IF SLD_CH_9_ACTIVE THEN SLD_TIME_TEMP[8] := SLD_CH_9.TIME_COUNT; END_IF

(*SLD_CH_10: AMS增压器滑油出口温度高降速*)
SLD_CH_10(FAILURE := AMS_TURBOCHG_OIL_TEMP_HIGH_SLD_P AND (NOT AMS_TURBOCHG_OIL_TEMP_HIGH_SLD_PASS_FAIL),
				T_FILTER := Slowdown_from_AMS_SHD_time_filter,
				T_DELAY  := Slowdown_from_AMS_SHD_time_delay,
				OVERRIDE := SLD_OVERRIDE);
AMS_TURBOCHG_OIL_TEMP_HIGH := SLD_CH_10.LED;
SLD_LAMP_OUT        := SLD_LAMP_OUT OR SLD_CH_10.LAMP;
SLD_SIGN_OUT        := SLD_SIGN_OUT OR SLD_CH_10.SIGN;
HORN_OUT            := HORN_OUT OR SLD_CH_10.HORN;
NORMAL_SLD_LAMP_OUT := NORMAL_SLD_LAMP_OUT OR SLD_CH_10.LAMP;
NORMAL_SLD_SIGN_OUT := NORMAL_SLD_SIGN_OUT OR SLD_CH_10.SIGN;
SLD_CH_10_ACTIVE := SLD_CH_10.FILTER_FAILURE_OUT;
IF SLD_CH_10_ACTIVE THEN SLD_TIME_TEMP[9] := SLD_CH_10.TIME_COUNT; END_IF

(*SLD_CH_11: AMS缸排气温度高降速*)
SLD_CH_11(FAILURE := AMS_CYL_EXHAUST_TEMP_HIGH_SLD_P AND (NOT AMS_CYL_EXHAUST_TEMP_HIGH_SLD_PASS_FAIL),
				T_FILTER := Slowdown_from_AMS_SHD_time_filter,
				T_DELAY  := Slowdown_from_AMS_SHD_time_delay,
				OVERRIDE := SLD_OVERRIDE);
AMS_CYL_EXHAUST_TEMP_HIGH := SLD_CH_11.LED;
SLD_LAMP_OUT        := SLD_LAMP_OUT OR SLD_CH_11.LAMP;
SLD_SIGN_OUT        := SLD_SIGN_OUT OR SLD_CH_11.SIGN;
HORN_OUT            := HORN_OUT OR SLD_CH_11.HORN;
NORMAL_SLD_LAMP_OUT := NORMAL_SLD_LAMP_OUT OR SLD_CH_11.LAMP;
NORMAL_SLD_SIGN_OUT := NORMAL_SLD_SIGN_OUT OR SLD_CH_11.SIGN;
SLD_CH_11_ACTIVE := SLD_CH_11.FILTER_FAILURE_OUT;
IF SLD_CH_11_ACTIVE THEN SLD_TIME_TEMP[10] := SLD_CH_11.TIME_COUNT; END_IF

(*SLD_CH_12: AMS增压器进口排气温度高降速*)
SLD_CH_12(FAILURE := AMS_TURBOCHG_INLET_EXHAUST_TEMP_HIGH_SLD_P AND (NOT AMS_TURBOCHG_INLET_EXHAUST_TEMP_HIGH_SLD_PASS_FAIL),
				T_FILTER := Slowdown_from_AMS_SHD_time_filter,
				T_DELAY  := Slowdown_from_AMS_SHD_time_delay,
				OVERRIDE := SLD_OVERRIDE);
AMS_TURBOCHG_INLET_EXHAUST_TEMP_HIGH := SLD_CH_12.LED;
SLD_LAMP_OUT        := SLD_LAMP_OUT OR SLD_CH_12.LAMP;
SLD_SIGN_OUT        := SLD_SIGN_OUT OR SLD_CH_12.SIGN;
HORN_OUT            := HORN_OUT OR SLD_CH_12.HORN;
NORMAL_SLD_LAMP_OUT := NORMAL_SLD_LAMP_OUT OR SLD_CH_12.LAMP;
NORMAL_SLD_SIGN_OUT := NORMAL_SLD_SIGN_OUT OR SLD_CH_12.SIGN;
SLD_CH_12_ACTIVE := SLD_CH_12.FILTER_FAILURE_OUT;
IF SLD_CH_12_ACTIVE THEN SLD_TIME_TEMP[11] := SLD_CH_12.TIME_COUNT; END_IF

(*SLD_CH_13: AMS缸扫气箱着火温度高降速*)
SLD_CH_13(FAILURE := AMS_SCAV_BOX_FIRE_TEMP_HIGH_SLD_P AND (NOT AMS_SCAV_BOX_FIRE_TEMP_HIGH_SLD_PASS_FAIL),
				T_FILTER := Slowdown_from_AMS_SHD_time_filter,
				T_DELAY  := Slowdown_from_AMS_SHD_time_delay,
				OVERRIDE := SLD_OVERRIDE);
AMS_SCAV_BOX_FIRE_TEMP_HIGH := SLD_CH_13.LED;
SLD_LAMP_OUT        := SLD_LAMP_OUT OR SLD_CH_13.LAMP;
SLD_SIGN_OUT        := SLD_SIGN_OUT OR SLD_CH_13.SIGN;
HORN_OUT            := HORN_OUT OR SLD_CH_13.HORN;
NORMAL_SLD_LAMP_OUT := NORMAL_SLD_LAMP_OUT OR SLD_CH_13.LAMP;
NORMAL_SLD_SIGN_OUT := NORMAL_SLD_SIGN_OUT OR SLD_CH_13.SIGN;
SLD_CH_13_ACTIVE := SLD_CH_13.FILTER_FAILURE_OUT;
IF SLD_CH_13_ACTIVE THEN SLD_TIME_TEMP[12] := SLD_CH_13.TIME_COUNT; END_IF

(*SLD_CH_14: 注油器断流降速*)
SLD_CH_14(FAILURE := LUBRICATOR_OIL_FLOW_FAIL_SLD_P AND (NOT LUBRICATOR_OIL_FLOW_FAIL_SLD_PASS_FAIL),
				T_FILTER := Lubricator_oil_flow_SLD_time_filter,
				T_DELAY  := Lubricator_oil_flow_SLD_time_delay,
				OVERRIDE := SLD_OVERRIDE);
LUBRICATOR_OIL_FLOW_FAIL := SLD_CH_14.LED;
SLD_LAMP_OUT        := SLD_LAMP_OUT OR SLD_CH_14.LAMP;
SLD_SIGN_OUT        := SLD_SIGN_OUT OR SLD_CH_14.SIGN;
HORN_OUT            := HORN_OUT OR SLD_CH_14.HORN;
NORMAL_SLD_LAMP_OUT := NORMAL_SLD_LAMP_OUT OR SLD_CH_14.LAMP;
NORMAL_SLD_SIGN_OUT := NORMAL_SLD_SIGN_OUT OR SLD_CH_14.SIGN;
SLD_CH_14_ACTIVE := SLD_CH_14.FILTER_FAILURE_OUT;
IF SLD_CH_14_ACTIVE THEN SLD_TIME_TEMP[13] := SLD_CH_14.TIME_COUNT; END_IF

(*SLD_CH_15: 调速器系统异常降速*)
SLD_CH_15(FAILURE := GOVERNOR_SYS_FAULT_SLD_P AND (NOT GOVERNOR_SYS_FAULT_SLD_PASS_FAIL),
				T_FILTER := Governor_sys_fault_SLD_time_filter,
				T_DELAY  := Governor_sys_fault_SLD_time_delay,
				OVERRIDE := SLD_OVERRIDE);
GOVERNOR_SYS_FAULT := SLD_CH_15.LED;
SLD_LAMP_OUT        := SLD_LAMP_OUT OR SLD_CH_15.LAMP;
SLD_SIGN_OUT        := SLD_SIGN_OUT OR SLD_CH_15.SIGN;
HORN_OUT            := HORN_OUT OR SLD_CH_15.HORN;
NORMAL_SLD_LAMP_OUT := NORMAL_SLD_LAMP_OUT OR SLD_CH_15.LAMP;
NORMAL_SLD_SIGN_OUT := NORMAL_SLD_SIGN_OUT OR SLD_CH_15.SIGN;
SLD_CH_15_ACTIVE := SLD_CH_15.FILTER_FAILURE_OUT;
IF SLD_CH_15_ACTIVE THEN SLD_TIME_TEMP[14] := SLD_CH_15.TIME_COUNT; END_IF

(*===========预期信号聚合, 合成 SHD/SLD_EXPTED_TO_UNIC 并写入全局变量===========*)
SHD_EXPTED_TO_UNIC :=
	SHD_CH_1_ACTIVE OR SHD_CH_2_ACTIVE OR SHD_CH_3_ACTIVE OR
	SHD_CH_4_ACTIVE OR SHD_CH_5_ACTIVE OR SHD_CH_6_ACTIVE;

SLD_EXPTED_TO_UNIC :=
	SLD_CH_1_ACTIVE  OR SLD_CH_2_ACTIVE  OR SLD_CH_3_ACTIVE  OR
	SLD_CH_4_ACTIVE  OR SLD_CH_5_ACTIVE  OR SLD_CH_6_ACTIVE  OR
	SLD_CH_7_ACTIVE  OR SLD_CH_8_ACTIVE  OR SLD_CH_9_ACTIVE  OR
	SLD_CH_10_ACTIVE OR SLD_CH_11_ACTIVE OR SLD_CH_12_ACTIVE OR
	SLD_CH_13_ACTIVE OR SLD_CH_14_ACTIVE OR SLD_CH_15_ACTIVE;

(*===========HMI 剩余延时最小值，写入全局 H_SHD/SLD_TIME_COUNT===========*)
IF SHD_EXPTED_TO_UNIC THEN
	TEMP_SHD_MIN := 200000;
	FOR x := 0 TO 5 DO
		IF SHD_TIME_TEMP[x] < TEMP_SHD_MIN THEN
			TEMP_SHD_MIN := SHD_TIME_TEMP[x];
			a := x;
		END_IF
	END_FOR
END_IF
IF NOT SHD_EXPTED_TO_UNIC OR SHD_OVERRIDE THEN
	H_SHD_TIME_COUNT := 0;
ELSE
	H_SHD_TIME_COUNT := SHD_TIME_TEMP[a] / 1000;
END_IF

IF SLD_EXPTED_TO_UNIC THEN
	TEMP_SLD_MIN := 200000;
	FOR y := 0 TO 14 DO
		IF SLD_TIME_TEMP[y] < TEMP_SLD_MIN THEN
			TEMP_SLD_MIN := SLD_TIME_TEMP[y];
			b := y;
		END_IF
	END_FOR
END_IF
IF NOT SLD_EXPTED_TO_UNIC OR SLD_OVERRIDE OR OMD_SLD_OVERRIDE THEN
	H_SLD_TIME_COUNT := 0;
ELSE
	H_SLD_TIME_COUNT := SLD_TIME_TEMP[b] / 1000;
END_IF
END_FUNCTION_BLOCK

(* POU SLD_SHD_PROCESS, ST *)
(*4.1.6.4*)
FUNCTION_BLOCK SLD_SHD_PROCESS
VAR_INPUT
	FAILURE: BOOL;
	OVERRIDE: BOOL;
	T_FILTER :TIME;
	T_DELAY :TIME;
END_VAR
VAR_OUTPUT
	LED: BOOL;
	HORN: BOOL;
	SIGN: BOOL;
	LAMP: BOOL;
      TIME_COUNT: REAL;
	FILTER_FAILURE_OUT:	BOOL;
END_VAR
VAR
	TONInst_FILTER: TON;
	TONInst_DELAY: TON;

	DELAY_FAILURE: BOOL;(*after time delay*)
	FILTER_FAILURE: BOOL;(*after timefilter*)

	SR_RINPUT: BOOL; (* SR FilpFlop Input*)
	OVERRIDE_RESET: BOOL;(*OR with RESET*)
	SR_OUTPUT: BOOL;

	TIMEET:TIME;(*INTERNAL TIME TRANSFER*)

	SRinst: SR;
END_VAR
(*INIT  VAR*)
DELAY_FAILURE := FALSE;(*after time delay*)
FILTER_FAILURE := FALSE;(*after timefilter*)

SR_RINPUT := FALSE; (* SR FilpFlop Input*)
OVERRIDE_RESET := FALSE;(*OR with RESET*)
SR_OUTPUT := FALSE;

(**INPUT Logic**)
TONInst_FILTER(IN := FAILURE, PT := T_FILTER);
FILTER_FAILURE := TONInst_FILTER.Q;

TONInst_DELAY(IN := FILTER_FAILURE, PT := T_DELAY);
DELAY_FAILURE :=	TONInst_DELAY.Q;

OVERRIDE_RESET :=	OVERRIDE OR RESET_SIGNAL;

SR_RINPUT := NOT DELAY_FAILURE AND OVERRIDE_RESET;

(*get SR OUTPUT*)
SRinst(SET1 := DELAY_FAILURE, RESET := SR_RINPUT);
SR_OUTPUT := SRinst.Q1;

(**OUTPUT**)
(* LED OUTPUT*)
LED := FAILURE OR SR_OUTPUT;

(*HORN   symbol '>' ??*)
HORN := SR_OUTPUT OR FILTER_FAILURE;

(*SIGN*)
SIGN := SR_OUTPUT AND (NOT OVERRIDE);


(*LAMP*)
LAMP := SR_OUTPUT OR (FILTER_FAILURE AND FLASHER_BLINK.OUT);


(*FILTER_FAILURE_OUT*)
FILTER_FAILURE_OUT  :=  FILTER_FAILURE;

(*DELAY TIME COUNT OUT*)
TIMEET:=TONInst_DELAY.PT-TONInst_DELAY.ET;
TIME_COUNT:= TIME_TO_REAL  (TIMEET);
END_FUNCTION_BLOCK

(* POU SWITCHES_ETC, ST *)
(*get SLD,SHD override status*)
FUNCTION_BLOCK  SWITCHES_ETC
VAR_INPUT
END_VAR
VAR_OUTPUT
END_VAR
VAR
	SR_Ins: SR;
	SR_IN1: BOOL;
	SR_IN2: BOOL;
	SR_TiltIN: BOOL;

	(*Flasher frequency change flag*)
	Frequency_Change_Flag: BOOL;
	FLASHER_FREQUENCY_OLD: REAL;

	(*R-TRIGGER for SHD_OVERRIDE_MAN_BX7331C*)
	R_TRIG_SHD_OVERRIDE_MAN: R_TRIG;
	(*R-TRIGGER for SHD_OVERRIDE_MAN_BX7331C*)
	R_TRIG_SHD_OVERRIDE_ECR_AUT: R_TRIG;
	(*timer for dynamic input of SHD_OVERRIDE_ECR_AUT*)

	(*SHUTDOWN OVERRIDER  判断输入信号之前状态是否为FALSE标志*)
	SHD_OVERRIDE_BR_FLAG:  BOOL;
	SHD_OVERRIDE_ECR_AUT_FLAG:  BOOL;
	(*自锁处理后的输入信号*)
	SHD_OVERRIDE_BR_SIGNAL:	BOOL;
	SHD_OVERRIDE_ECR_AUT_SIGNAL:  BOOL;

	(*OMD SLD OVERRIDER  判断输入信号之前状态是否为FALSE标志*)
	SLD_OMD_OVERRIDE_BR_FLAG:  BOOL;
	SLD_OMD_OVERRIDE_ECR_AUT_FLAG:  BOOL;
	(*自锁处理后的输入信号*)
	SLD_OMD_OVERRIDE_BR_SIGNAL:	BOOL;
	SLD_OMD_OVERRIDE_ECR_AUT_SIGNAL:  BOOL;

	(*SLD OVERRIDER  判断输入信号之前状态是否为FALSE标志*)
	SLD_OVERRIDE_BR_FLAG:  BOOL;
	SLD_OVERRIDE_ECR_AUT_FLAG:  BOOL;
	(*自锁处理后的输入信号*)
	SLD_OVERRIDE_BR_SIGNAL:	BOOL;
	SLD_OVERRIDE_ECR_AUT_SIGNAL:  BOOL;


	(*BR CENTER  3 pushButton  判断输入信号之前状态是否为FALSE标志 *)
	BR_CENTERL_SLD_FLAG:  BOOL;
	BR_CENTERL_OMD_SLD_FLAG:  BOOL;
	BR_CENTERL_SHD_FLAG:  BOOL;
	(*自锁处理后的输入信号*)
	BR_CENTERL_SLD_SIGNAL:	BOOL;
	BR_CENTERL_OMD_SLD_SIGNAL:  BOOL;
	BR_CENTERL_SHD_SIGNAL:  BOOL;

	(*BR PORT  3 pushButton  判断输入信号之前状态是否为FALSE标志 *)
	BR_PORT_SLD_FLAG:  BOOL;
	BR_PORT_OMD_SLD_FLAG:  BOOL;
	BR_PORT_SHD_FLAG:  BOOL;
	(*自锁处理后的输入信号*)
	BR_PORT_SLD_SIGNAL:	BOOL;
	BR_PORT_OMD_SLD_SIGNAL:  BOOL;
	BR_PORT_SHD_SIGNAL:  BOOL;

	(*BR STBD  3 pushButton  判断输入信号之前状态是否为FALSE标志 *)
	BR_STBD_SLD_FLAG:  BOOL;
	BR_STBD_OMD_SLD_FLAG:  BOOL;
	BR_STBD_SHD_FLAG:  BOOL;
	(*自锁处理后的输入信号*)
	BR_STBD_SLD_SIGNAL:	BOOL;
	BR_STBD_OMD_SLD_SIGNAL:  BOOL;
	BR_STBD_SHD_SIGNAL:  BOOL;






	HZ_INT: INT;
	TIMEHZ: REAL;
END_VAR
(*INIT  VAR*)
SR_IN1 := FALSE;
SR_IN2 := FALSE;
SR_TiltIN := FALSE;


(******************** BR CENTER ********************)
IF	BR_CENTER_CANCEL_SLD_P = TRUE
THEN
	IF	BR_CENTERL_SLD_FLAG = FALSE    
	THEN
		(*信号反转*)
		BR_CENTERL_SLD_SIGNAL := NOT	BR_CENTERL_SLD_SIGNAL;

		BR_CENTERL_SLD_FLAG := TRUE;
	END_IF
ELSE
	BR_CENTERL_SLD_FLAG	:=	FALSE;
END_IF


IF	BR_CENTER_CANCEL_OMD_SLD_P = TRUE
THEN
	IF	BR_CENTERL_OMD_SLD_FLAG = FALSE
	THEN
		(*信号反转*)
		BR_CENTERL_OMD_SLD_SIGNAL := NOT	BR_CENTERL_OMD_SLD_SIGNAL;

